// TIA Portal project "Tunel_Paster_16000" (V16)

(* hardware
DEVICE "S7-1200 station_1"  S7-1200 Station
   slot 0: "Rack_0"  S7-1200 Rack  Rack  V1.0
   slot 1: "PLC_1"  CPU 1215C AC/DC/Rly  6ES7 215-1BG40-0XB0  V4.4
*)

// ===== PLC "PLC_1"  CPU 1215C AC/DC/Rly =====

VAR_GLOBAL   // PLC tag table "Default tag table"
   "bStateZones_OK" AT %M10.0 : Bool;   // Все зоны готовы к работе
   "bHasPrior_Stop" AT %M10.1 : Bool;   // Имеется маркер разрешения "СТОП - конвейер
   "bStart_Main_TunelPaster" AT %M1.7 : Bool;   // Старт-Работа тунельного пастеризатора (ОБЩИЙ)
   "bMain_AlarmSystem" AT %M2.3 : Bool;   // АВария в системе (Общая)
   "iNomberZoneAlarm" AT %MW6 : Int;   // Номер зоны с отклонениями
   "Разрешение работы конвейера" AT %M0.0 : Bool;   // Команда разрешения от Глобального блока работы
   "Авария, ошибка в системе" AT %M0.1 : Bool;   // Метка ошибок или аварий
   "Clock_Byte" AT %MB500 : Byte;
   "Clock_10Hz" AT %M500.0 : Bool;
   "Clock_5Hz" AT %M500.1 : Bool;
   "Clock_2.5Hz" AT %M500.2 : Bool;
   "Clock_2Hz" AT %M500.3 : Bool;
   "Clock_1.25Hz" AT %M500.4 : Bool;
   "Clock_1Hz" AT %M500.5 : Bool;
   "Clock_0.625Hz" AT %M500.6 : Bool;
   "Clock_0.5Hz" AT %M500.7 : Bool;
END_VAR

VAR_GLOBAL   // PLC tag table "HMI_"
   "bHMI_button_Start" AT %M2.0 : Bool;   // Кнопка старт
   "bHMI_button_Stop" AT %M2.1 : Bool;   // Кнопка стоп
   "bHMI_button_Pause" AT %M2.2 : Bool;   // Кнопка пауза
   "bHMI_Button_ConveyorStart" AT %M2.4 : Bool;   // Кнопка подтверждения старта конвейера
   "bStartAllowed" AT %M100.0 : Bool;   // Готовность к старту
   "bOpenWindStartConveyor" AT %M100.1 : Bool;   // Вызов окна подтверждения оператором старта конвейера
   "bHMI_ResetAlarm" AT %M0.2 : Bool;   // Сброс аварий
   "iHMI_Num_StatrPaster" AT %MW4 : Int;
   "sHMI_Text_State" AT %MB3 : Char;   // Ткстом статус пастеризатора
   "bTypePID_Zone1" AT %M8.0 : Bool;   // Тип ПИД - 1 - Охлаждение, 0 - Нагрев
   "bTypePID_Zone2" AT %M8.1 : Bool;   // Тип ПИД - 1 - Охлаждение, 0 - Нагрев
   "bTypePID_Zone3" AT %M8.2 : Bool;   // Тип ПИД - 1 - Охлаждение, 0 - Нагрев
   "bTypePID_Zone4" AT %M8.3 : Bool;   // Тип ПИД - 1 - Охлаждение, 0 - Нагрев
   "bTypePID_Zone5" AT %M8.4 : Bool;   // Тип ПИД - 1 - Охлаждение, 0 - Нагрев
END_VAR

VAR_GLOBAL   // PLC tag table "DI"
   "xAlarm_StopButton" AT %I2.0 : Bool;   // Физическая Кнопка стоп
   "xAlarmPump_1" AT %I2.1 : Bool;   // СИгнал аварии от насоса
   "xAlarmPump_2" AT %I2.2 : Bool;   // СИгнал аварии от насоса
   "xAlarmPump_3" AT %I2.3 : Bool;   // СИгнал аварии от насоса
   "xAlarmPump_4" AT %I2.4 : Bool;   // СИгнал аварии от насоса
   "xAlarmPump_5" AT %I2.5 : Bool;   // СИгнал аварии от насоса
   "xAlarmPump_6" AT %I2.6 : Bool;   // СИгнал аварии от насоса
   "xAlarmPump_7" AT %I2.7 : Bool;   // СИгнал аварии от насоса
END_VAR

VAR_GLOBAL   // PLC tag table "Test_PID"
   "set" AT %MD30 : Real;
   "in" AT %MD34 : Real;
   "MAnual" AT %M38.0 : Bool;
   "MValue" AT %MD40 : Real;
   "rOut" AT %MD46 : Real;
   "Mode" AT %MW44 : Int;
   "ResPID" AT %M50.0 : Bool;
END_VAR

VAR_GLOBAL   // PLC tag table "MyTags"
   "InTempZone1" AT %MD12 : Real;   // Зона 1 - температура - обработанная
   "InTempZone2" AT %MD16 : Real;   // Зона 2 - температура - обработанная
   "InTempZone3" AT %MD20 : Real;   // Зона 3 - температура - обработанная
   "InTempZone4" AT %MD24 : Real;   // Зона 4 - температура - обработанная
   "InTempZone5" AT %MD28 : Real;   // Зона 5 - температура - обработанная
END_VAR

TYPE "FV_o/c"
   STRUCT
      bOpenCmd : Bool;   // Команда открыть (автомат)
      bManualMode : Bool;   // Ручной режим (TRUE)
      bManualOpen : Bool;   // Команда открыть в ручном режиме
      bFeedbackOpen : Bool;   // Обратная связь "Открыт"
      tMaxTime : Time;   // Время на открытие
      bResetAlarm : Bool;   // Сброс аварии
      bCheckFeedback : Bool;   // Выбирается есть ли обратная связь у клапана
      bOutOpen : Bool;   // Выход на открытие клапана
      iOutState : Int;   // Выход статуса клапана
      bOutFault : Bool;   // Выход ошибки клапана
   END_STRUCT;
END_TYPE

TYPE "ZoneStatus"
   STRUCT
      bInSetpoint : Bool;   // Зона в уставке по температуре
      bOutOfRange : Bool;   // Зона вышла от уставки на > дельта
      bHasPriority : Bool;   // Зона имеет приоритет на остановку конвейера
   END_STRUCT;
END_TYPE

TYPE "Zone_Pararm"
   STRUCT
      rTemp : Real;   // Температура с датчика
      rSet : Real;   // Уставка
      rDelta : Real;   // Дельта
      bPriority : Bool;   // Приоритет
      bOUT_ZoneStatus : "ZoneStatus";   // Состояние зоны_
   END_STRUCT;
END_TYPE

TYPE "FV_regul"
   STRUCT
      bHMI_ManualMode : Bool;   // Переключение режима авто/ручно (0 - А, 1 - Р)
      rHMI_ManualSet : Real;   // Уставка в ручном режиме (0-100)
      rAuto_Set : Real;   // Уставка в автоматическом режиме
      iOut_AO : Int;   // Сигнал на аналоговый выход
      "rHMI_Out_FV-%" : Real;   // Состояние в % (0-100)
      bOut_DO_ValveOpen : Bool;   // Дискретный сигнал открытия
   END_STRUCT;
END_TYPE

TYPE "Коэф ПИД"
   STRUCT
      Gain : Int;   // Коэф П
      I : DInt;   // Коэф И
      D : DInt;   // Коэф Д
   END_STRUCT;
END_TYPE

TYPE "PE_Param"
   STRUCT
      rСкоростьКонвейера : Real;
      rПЕ_Задан : Real;
      rДлина_Конв : Real;
      rZ_Коэф : Real := 1.393;
      rТref : Real := 60.0;
      rТемп_Мин : Real;
      rТемп_Макс : Real;
      "rСкоростьКонв_м/с" : Real;
      rРучноеЗначТемп : Real;
      diВремяПростоя : DInt := 60000;
      bManualTemp : Bool;
   END_STRUCT;
END_TYPE

// folder: DB-FB

DATA_BLOCK "FB_check_For_Start_DB"   // DB1
{ S7_Optimized_Access := 'FALSE' }
VERSION : 0.1
// stored: InstanceOfName FB_check_For_Start
"FB_check_For_Start"
BEGIN
END_DATA_BLOCK

DATA_BLOCK "FB_Emergency_DB"   // DB3
{ S7_Optimized_Access := 'FALSE' }
VERSION : 0.1
// stored: InstanceOfName -FB_Emergency
"-FB_Emergency"
BEGIN
END_DATA_BLOCK

DATA_BLOCK "FB_CheckZoneStatus_DB"   // DB11
{ S7_Optimized_Access := 'FALSE' }
VERSION : 0.1
// stored: InstanceOfName FB_CheckZoneStatus
"FB_CheckZoneStatus"
BEGIN
END_DATA_BLOCK

DATA_BLOCK "FB_Управление конвейером_DB"   // DB18
{ S7_Optimized_Access := 'FALSE' }
VERSION : 0.1
// stored: InstanceOfName FB_Управление конвейером
"FB_Управление конвейером"
BEGIN
END_DATA_BLOCK

DATA_BLOCK "FB_GlobalStateManager_DB"   // DB31
{ S7_Optimized_Access := 'FALSE' }
VERSION : 0.1
// stored: InstanceOfName FB_GlobalStateManager
"FB_GlobalStateManager"
BEGIN
END_DATA_BLOCK

DATA_BLOCK "FB_PE_Control_DB"   // DB38
{ S7_Optimized_Access := 'TRUE' }
VERSION : 0.1
// stored: InstanceOfName FB_PE_Control
"FB_PE_Control"
BEGIN
END_DATA_BLOCK

// folder: Use VARs to HMI

DATA_BLOCK "DB2_HMI_SET"   // DB2
{ S7_Optimized_Access := 'FALSE' }
VERSION : 0.1
   VAR
      dwSetMinOutDelta : DInt;   // Время ожидания при выходе за пределы уставок
      dwSetMinInDelta : DInt;   // Время ожидания при возврате к уставкам
      dwSetTimeWaitToStart : DInt;   // Время ожидания выхода на режим пастеризатора
      "dwВремя ожидания_стабилизации_темп" : DInt;   // Вреямя ожидания стабилизации температур при выходе за пределы
      rSetTemp_Zone1 : Real;   // Уставка температуры зоны 1
      rSetTemp_Zone2 : Real;   // Уставка температуры зоны 2
      rSetTemp_Zone3 : Real;   // Уставка температуры зоны 3
      rSetTemp_Zone4 : Real;   // Уставка температуры зоны 4
      rSetTemp_Zone5 : Real;   // Уставка температуры зоны 5
      k_PID_Zona1 : "Коэф ПИД";   // ПИД - ЗОна 1
      k_PID_Zona2 : "Коэф ПИД";   // ПИД - зона 2
      k_PID_Zona3 : "Коэф ПИД";   // ПИД - ЗОна 3
      k_PID_Zona4 : "Коэф ПИД";   // ПИД - зона 4
      k_PID_Zona5 : "Коэф ПИД";   // ПИД - ЗОна 5
      HMI_PE : "PE_Param";
   END_VAR
BEGIN
   k_PID_Zona1.Gain := 1;
   k_PID_Zona1.I := 20;
   k_PID_Zona2.Gain := 1;
   k_PID_Zona2.I := 20;
   k_PID_Zona3.Gain := 1;
   k_PID_Zona3.I := 20;
   k_PID_Zona4.Gain := 1;
   k_PID_Zona4.I := 20;
   k_PID_Zona5.Gain := 1;
   k_PID_Zona5.I := 20;
END_DATA_BLOCK

DATA_BLOCK "FVs_o/p"   // DB6
{ S7_Optimized_Access := 'FALSE' }
VERSION : 0.1
   VAR
      FV_1 : "FV_o/c";
      FV_2 : "FV_o/c";
      FV_3 : "FV_o/c";
      FV_4 : "FV_o/c";
      FV_5 : "FV_o/c";
      FV_6 : "FV_o/c";
      FV_7 : "FV_o/c";
   END_VAR
BEGIN
END_DATA_BLOCK

DATA_BLOCK "Zones_Param"   // DB15
{ S7_Optimized_Access := 'FALSE' }
VERSION : 0.1
   VAR
      Zone_1_Преднагрев : "Zone_Pararm";
      Zone_2_Нагрев : "Zone_Pararm";
      Zone_3_Пастеризация : "Zone_Pararm";
      Zone_4_Охлаждение1 : "Zone_Pararm";
      Zone_5_Охлаждение2 : "Zone_Pararm";
   END_VAR
BEGIN
END_DATA_BLOCK

DATA_BLOCK "FVs_Regul"   // DB24
{ S7_Optimized_Access := 'FALSE' }
VERSION : 0.1
   VAR
      FV_Regul_1 : "FV_regul";
      FV_Regul_2 : "FV_regul";
      FV_Regul_3 : "FV_regul";
      FV_Regul_4 : "FV_regul";
      FV_Regul_5 : "FV_regul";
   END_VAR
BEGIN
END_DATA_BLOCK

DATA_BLOCK "Pumps"   // DB30
{ S7_Optimized_Access := 'FALSE' }
VERSION : 0.1
BEGIN
END_DATA_BLOCK

// folder: Зоны/DB_Zone

DATA_BLOCK "FB_Zone_Control_1_Преднагрев_DB"   // DB12
{ S7_Optimized_Access := 'FALSE' }
VERSION : 0.1
// stored: InstanceOfName FB_Zone_Control
"FB_Zone_Control"
BEGIN
END_DATA_BLOCK

DATA_BLOCK "FB_Zone_Control_2_Нагрев_DB"   // DB13
{ S7_Optimized_Access := 'FALSE' }
VERSION : 0.1
// stored: InstanceOfName FB_Zone_Control
"FB_Zone_Control"
BEGIN
END_DATA_BLOCK

DATA_BLOCK "FB_Zone_Control_3_Пастеризация_DB"   // DB14
{ S7_Optimized_Access := 'FALSE' }
VERSION : 0.1
// stored: InstanceOfName FB_Zone_Control
"FB_Zone_Control"
BEGIN
END_DATA_BLOCK

DATA_BLOCK "FB_Zone_Control_4_Охлаждение_DB"   // DB16
{ S7_Optimized_Access := 'FALSE' }
VERSION : 0.1
// stored: InstanceOfName FB_Zone_Control
"FB_Zone_Control"
BEGIN
END_DATA_BLOCK

DATA_BLOCK "FB_Zone_Control_5_Охлаждение2_DB"   // DB17
{ S7_Optimized_Access := 'FALSE' }
VERSION : 0.1
// stored: InstanceOfName FB_Zone_Control
"FB_Zone_Control"
BEGIN
END_DATA_BLOCK

// folder: Клапана/FV_o/C/FV_DB

DATA_BLOCK "FV_1"   // DB4
{ S7_Optimized_Access := 'FALSE' }
VERSION : 0.1
// stored: InstanceOfName Valve(c/o)
"Valve(c/o)"
BEGIN
END_DATA_BLOCK

DATA_BLOCK "FV_5"   // DB5
{ S7_Optimized_Access := 'FALSE' }
VERSION : 0.1
// stored: InstanceOfName Valve(c/o)
"Valve(c/o)"
BEGIN
END_DATA_BLOCK

DATA_BLOCK "FV_6"   // DB7
{ S7_Optimized_Access := 'FALSE' }
VERSION : 0.1
// stored: InstanceOfName Valve(c/o)
"Valve(c/o)"
BEGIN
END_DATA_BLOCK

DATA_BLOCK "FV_7"   // DB8
{ S7_Optimized_Access := 'FALSE' }
VERSION : 0.1
// stored: InstanceOfName Valve(c/o)
"Valve(c/o)"
BEGIN
END_DATA_BLOCK

DATA_BLOCK "FV_2"   // DB9
{ S7_Optimized_Access := 'FALSE' }
VERSION : 0.1
// stored: InstanceOfName Valve(c/o)
"Valve(c/o)"
BEGIN
END_DATA_BLOCK

DATA_BLOCK "FV_3"   // DB10
{ S7_Optimized_Access := 'FALSE' }
VERSION : 0.1
// stored: InstanceOfName Valve(c/o)
"Valve(c/o)"
BEGIN
END_DATA_BLOCK

DATA_BLOCK "FV_4"   // DB19
{ S7_Optimized_Access := 'FALSE' }
VERSION : 0.1
// stored: InstanceOfName Valve(c/o)
"Valve(c/o)"
BEGIN
END_DATA_BLOCK

// folder: Клапана/FV_regul/DB

DATA_BLOCK "FV_Regul_1_DB"   // DB20
{ S7_Optimized_Access := 'FALSE' }
VERSION : 0.1
// stored: InstanceOfName Valve(regul)
"Valve(regul)"
BEGIN
END_DATA_BLOCK

DATA_BLOCK "FV_Regul_2_DB"   // DB21
{ S7_Optimized_Access := 'FALSE' }
VERSION : 0.1
// stored: InstanceOfName Valve(regul)
"Valve(regul)"
BEGIN
END_DATA_BLOCK

DATA_BLOCK "FV_Regul_3_DB"   // DB22
{ S7_Optimized_Access := 'FALSE' }
VERSION : 0.1
// stored: InstanceOfName Valve(regul)
"Valve(regul)"
BEGIN
END_DATA_BLOCK

DATA_BLOCK "FV_Regul_4_DB"   // DB23
{ S7_Optimized_Access := 'FALSE' }
VERSION : 0.1
// stored: InstanceOfName Valve(regul)
"Valve(regul)"
BEGIN
END_DATA_BLOCK

DATA_BLOCK "FV_Regul_5_DB"   // DB37
{ S7_Optimized_Access := 'FALSE' }
VERSION : 0.1
// stored: InstanceOfName Valve(regul)
"Valve(regul)"
BEGIN
END_DATA_BLOCK

// folder: Насосы/DB

DATA_BLOCK "Pump_1_DB"   // DB25
{ S7_Optimized_Access := 'FALSE' }
VERSION : 0.1
// stored: InstanceOfName Pump
"Pump"
BEGIN
END_DATA_BLOCK

DATA_BLOCK "Pump_2_DB"   // DB26
{ S7_Optimized_Access := 'FALSE' }
VERSION : 0.1
// stored: InstanceOfName Pump
"Pump"
BEGIN
END_DATA_BLOCK

DATA_BLOCK "Pump_5_DB"   // DB27
{ S7_Optimized_Access := 'FALSE' }
VERSION : 0.1
// stored: InstanceOfName Pump
"Pump"
BEGIN
END_DATA_BLOCK

DATA_BLOCK "Pump_4_DB"   // DB28
{ S7_Optimized_Access := 'FALSE' }
VERSION : 0.1
// stored: InstanceOfName Pump
"Pump"
BEGIN
END_DATA_BLOCK

DATA_BLOCK "Pump_3_DB"   // DB29
{ S7_Optimized_Access := 'FALSE' }
VERSION : 0.1
// stored: InstanceOfName Pump
"Pump"
BEGIN
END_DATA_BLOCK

// folder: (top level)

FUNCTION_BLOCK "Pump"   // FB1, SCL
{ S7_Optimized_Access := 'FALSE' }
VERSION : 0.1
   VAR_INPUT
      bManualMode : Bool;   // Выбор ручного режима
      bManualStart : Bool;   // Ручной режим - старт
      bManualStop : Bool;   // Ручной режим - стоп
      rManualSpeed : Real;   // Ручной режим - скорость
      bAutoStartPerm : Bool;   // Команда на работоу в авто режиме
      rAutoSpeed : Real;   // Скорость в авто режиме
      bDriveReady : Bool;   // Готовность привода (автоматы)
      bDriveRunning : Bool;   // Привод в работе
      bDriveFault : Bool;   // Привод в ошибке
      rMinSpeed : Real;   // Минимальная скорость
      rMaxSpeed : Real;   // Максимальная скорость
      bResetFault : Bool;   // Сброс аварии
   END_VAR
   VAR_OUTPUT
      bRunCmd : Bool;   // Пуск частотника
      "rSpeedHMI(0-100)" : Real;   // Скорость работы (0-100) для HMI
      iSpeedOut : Int;   // Скорость насоса для аналогового выхода
      bPumpRunning : Bool;   // Работа
      bPumpFault : Bool;   // Авария
      iStatus : Int;   // Статус (0 - стоп 1 - работа 2 - авария)
   END_VAR
   VAR
      bFaultLatch : Bool;
      bRunRequest : Bool;
      rSpeedPump : Real;   // Скорость насоса
   END_VAR
BEGIN
   // 1. Обработка аварий
   #bFaultLatch := (#bDriveFault OR #bFaultLatch) AND NOT #bResetFault;
   #bPumpFault := #bFaultLatch;

   // 2. Формирование команды "Пуск"
   IF #bManualMode THEN
       // Ручной режим
       IF #bManualStart AND NOT #bManualStop THEN
           #bRunRequest := TRUE;
       ELSIF #bManualStop OR NOT #bDriveReady THEN
           #bRunRequest := FALSE;
       END_IF;
   ELSE
       // Автоматический режим
       #bRunRequest := #bAutoStartPerm AND NOT #bDriveFault;
   END_IF;

   // 3. Задание скорости
   IF #bManualMode THEN
       #"rSpeedHMI(0-100)" := LIMIT(MN := #rMinSpeed, IN := #rManualSpeed, MX := #rMaxSpeed);
   ELSE
       #"rSpeedHMI(0-100)" := LIMIT(MN := #rMinSpeed, IN := #rAutoSpeed, MX := #rMaxSpeed);
   END_IF;

   // Преобразование значения от 0-100 до 0-27648 для аналогового выхода
   #iSpeedOut := REAL_TO_INT((#"rSpeedHMI(0-100)"/ 100.0) * 27648.0);

   // 4. Выходные команды и статусы
   #bRunCmd := #bRunRequest AND NOT #bFaultLatch AND #bDriveReady;
   #bPumpRunning := #bDriveRunning AND #bRunCmd;

   // 5. Числовой статус (для HMI/SCADA)
   IF #bFaultLatch THEN
       #iStatus := 2; // Авария
   ELSIF #bPumpRunning THEN
       #iStatus := 1; // Работа
   ELSE
       #iStatus := 0; // Стоп
   END_IF;
END_FUNCTION_BLOCK

FUNCTION_BLOCK "FB_GlobalStateManager"   // FB2, SCL
{ S7_Optimized_Access := 'FALSE' }
VERSION : 0.1
   VAR_INPUT
      bStartCmd : Bool;   // Команда на старт от HMI
      bConfirmStart : Bool;   // Подтверждение оператора
      bResetFault : Bool;   // Сброс ошибки
      bAllSetpointsReached : Bool;   // // Все температуры достигли уставок
      bNoFaults : Bool;   // Нет аварий
      tStartTimeout : Time := T#30m;   // Время за которое пастер выходит на режим
      tReadyDelay : Time := t#10s;   // Время ожидания при выходе на режим до готовности
   END_VAR
   VAR_OUTPUT
      eState : Int;   // Текущее состояние
      bConveyorEnable : Bool;   // Разрешение на работу конвейера
      bSystemReady : Bool;   // Готовность системы
      bSystemFault : Bool;   // Состояние Fault
      sStatusText : WString;   // Текст для HMI
   END_VAR
   VAR
      tonStartTimeout : TON_TIME;   // Таймер выхода на режим
      tonReadyDelay : TON_TIME;   // Таймер готовности
   END_VAR
   VAR CONSTANT
      cSTATE_IDLE : Int;
      cSTATE_CHECK : Int := 10;
      cSTATE_STARTING : Int := 20;
      cSTATE_READY_DELAY : Int := 30;
      cSTATE_READY : Int := 40;
      cSTATE_FAULT : Int := 99;
      sText1 : String := 'Waiting';
   END_VAR
BEGIN
   // Таймеры
   #tonStartTimeout(IN := (#eState = #cSTATE_STARTING) AND NOT #bAllSetpointsReached, PT := #tStartTimeout);

   #tonReadyDelay(IN := (#eState = #cSTATE_READY_DELAY), PT := #tReadyDelay);

   // Основной CASE
   CASE #eState OF

       #cSTATE_IDLE:
        //   #sStatusText := 'Ожидание команды старта';
           IF #bStartCmd THEN
               #eState := #cSTATE_CHECK;
           END_IF;

       #cSTATE_CHECK:
       //    #sStatusText := 'Проверка условий старта';
           IF NOT #bNoFaults THEN
               #eState := #cSTATE_FAULT;
           ELSE
               #eState := #cSTATE_STARTING;
           END_IF;

       #cSTATE_STARTING:
      //     #sStatusText := 'Выход на уставки';
           IF #bAllSetpointsReached THEN
               #eState := #cSTATE_READY_DELAY;
           ELSIF #tonStartTimeout.Q THEN
               #eState := #cSTATE_FAULT;
           END_IF;

       #cSTATE_READY_DELAY:
      //     #sStatusText := 'dfsf';
           IF #tonReadyDelay.Q THEN
               #eState := #cSTATE_READY_DELAY;
           END_IF;

       #cSTATE_READY_DELAY:
      //     #sStatusText := 'Готово, ожидание подтверждения';
           #bSystemReady := TRUE;
           IF #bConfirmStart THEN
               #bConveyorEnable := TRUE;
           END_IF;

       #cSTATE_FAULT:
     //      #sStatusText := 'Авария! Требуется сброс';
           #bSystemFault := TRUE;
           IF #bResetFault AND #bNoFaults THEN
               #eState := #cSTATE_IDLE;
           END_IF;

       ELSE
           #eState := #cSTATE_IDLE;

   END_CASE;
END_FUNCTION_BLOCK

FUNCTION_BLOCK "Valve(c/o)"   // FB3, SCL
{ S7_Optimized_Access := 'FALSE' }
VERSION : 0.1
   VAR_INPUT
      bAuto_OpenCmd : Bool;   // Команда открыть (автомат)
      bManualMode : Bool;   // Ручной режим (TRUE)
      bManualOpen : Bool;   // Команда открыть в ручном режиме
      bFeedbackOpen : Bool;   // Обратная связь "Открыт"
      tMaxTime : Time;   // Время на открытие
      bResetAlarm : Bool;   // Сброс аварии
      bHaveFeedback : Bool;   // Есть ли обратная связь (0 - нет, 1 есть)
   END_VAR
   VAR_OUTPUT
      bValveOpen : Bool;   // Управляющий выход
      iValveState : Int;   // 0 = Закрыт, 1 = Открыт, 2 = Авария
      bValveFault : Bool;   // Авария
   END_VAR
   VAR
      tiOpenTimer : TON_TIME;   // Таймер на открытие
      bWaitingOpen : Bool;   // Флаг ожидания открытия
      bEnableTimer : Bool;   // Флаг активации таймера
   END_VAR
BEGIN

   // Обновление таймера — всегда в одном месте, вне условий
   #tiOpenTimer(
                IN := #bEnableTimer,
                PT := #tMaxTime
   );

   // Сброс
   IF #bResetAlarm THEN
       #bValveFault := FALSE;
       #bWaitingOpen := FALSE;
       #bEnableTimer := FALSE;
   END_IF;

   // === Режим: РУЧНОЙ ===
   IF #bManualMode THEN
       #bValveOpen := #bManualOpen;
       #bValveFault := FALSE;          // Аварии в ручном режиме не учитываются
       #bEnableTimer := FALSE;
       #bWaitingOpen := FALSE;

       // === Режим: АВТО ===
   ELSE

           // Управление выходом с учетом аварии, с контролем обратной связи
        IF #bAuto_OpenCmd AND NOT #bValveFault THEN
                   #bValveOpen := TRUE;
        ELSE
                   #bValveOpen := FALSE;
               END_IF;

               //  Проверяем, есть ли контроль обратной связи
        IF #bHaveFeedback THEN
            // Контроль открытия
            IF #bAuto_OpenCmd AND NOT #bFeedbackOpen AND NOT #bValveFault THEN
                #bEnableTimer := TRUE;
                #bWaitingOpen := TRUE;
            ELSE
                #bEnableTimer := FALSE;
                ;
                IF #bFeedbackOpen THEN
                    #bWaitingOpen := FALSE;
                END_IF;
            END_IF;
        END_IF;


           // Авария
           IF #tiOpenTimer.Q AND #bWaitingOpen THEN
               #bValveFault := TRUE;
               #bWaitingOpen := FALSE;
           END_IF;

   END_IF;


   // Состояние клапана
   IF #bValveFault THEN
       #iValveState := 2;       // Авария
   ELSIF #bHaveFeedback AND #bFeedbackOpen  THEN
       #iValveState := 1;       // Открыт
   ELSIF NOT #bHaveFeedback AND (NOT #bManualMode AND #bAuto_OpenCmd) OR (#bManualOpen AND #bManualMode) THEN
       #iValveState := 1;       // Открыт 
   ELSE
       #iValveState := 0;       // Закрыт
   END_IF;
END_FUNCTION_BLOCK

FUNCTION_BLOCK "Valve(regul)"   // FB4, SCL
{ S7_Optimized_Access := 'FALSE' }
VERSION : 0.1
   VAR_INPUT
      bManualMode : Bool;   // TRUE = ручной режим, FALSE = автоматический режим
      rAutoSetpoint : Real;   // Уставка открытия клапана в % (0.0–100.0) в автомате
      rManualSetpoint : Real;   // Уставка открытия клапана в % (0.0–100.0) в ручном режиме
   END_VAR
   VAR_OUTPUT
      iAnalogOutput : Int;   // Значение для аналогового выхода (0–27648)
      rValvePosPercent : Real;   // Текущее % открытия клапана для HMI
      bValveOpen : Bool;   // Дискретный сигнал "клапан открыт" (TRUE, если >0%)
   END_VAR
   VAR
      rSetpointPercent : Real;   // Расчётная уставка % открытия в текущем режиме
   END_VAR
BEGIN
       // Выбор уставки в зависимости от режима
       IF #bManualMode THEN
           #rSetpointPercent := #rManualSetpoint;
       ELSE
           #rSetpointPercent := #rAutoSetpoint;
       END_IF;

       // Ограничение % от 0.0 до 100.0
       IF #rSetpointPercent < 0.0 THEN
           #rSetpointPercent := 0.0;
       ELSIF #rSetpointPercent > 100.0 THEN
           #rSetpointPercent := 100.0;
       END_IF;

       // Перевод % в значение для аналогового выхода
       #iAnalogOutput := REAL_TO_INT((#rSetpointPercent / 100.0) * 27648.0);

           // Вывод значения для HMI
       #rValvePosPercent := #rSetpointPercent;

       // Дискретный сигнал "клапан открыт", если % > 0
       #bValveOpen := #rSetpointPercent > 0.0;
END_FUNCTION_BLOCK

FUNCTION_BLOCK "FB_Управление конвейером"   // FB5, SCL
{ S7_Optimized_Access := 'FALSE' }
VERSION : 0.1
   VAR_INPUT
      bEnable : Bool;   // Общий флаг работы системы
      bStartCmd : Bool;   // Команда на запуск от HMI, по кнопке из окна подтверждения
      bAllZonesInSetpoint : Bool;   // Все зоны достигли уставок
      bGlobalFault : Bool;   // Авария по системе
      bZoneHasPriority : Bool;   // У зоны с отклонением есть приоритет
      dwDeltaTempDelayMin : DWord;   // Задержка (мин), прежде чем остановить конвейер при отклонении
      dwResumeDelayMin : DInt;   // Время возврата после нормализации
   END_VAR
   VAR_OUTPUT
      bConveyorRun : Bool;   // Команда на пуск частотников
      bReadyToStart : Bool;   // Готовность к работе конвейера
      bWaitingConfirm : Bool;   // Ждём подтверждения от оператора, вывод окна на HMI
      bPaused : Bool;   // Конвейер остановлен по отклонению
   END_VAR
   VAR
      bStarted : Bool;   // Внутреннее состояние — процесс стартовал
      tiPauseTimer : TON_TIME;   // Таймер задержки перед остановкой
      tiResumeTimer : TON_TIME;   // Таймер ожидания перед возобновлением
      aZoneS_Status : Array[1..5] of "ZoneStatus";   // Массив для сбора состояния зон
      i : Int;
   END_VAR
   // tiPauseTimer.PT := T#1s;
   // tiResumeTimer.PT := T#1s;
BEGIN

   // Проверка на наличие флага обей работы системы
   IF NOT #bEnable THEN
       #bReadyToStart := FALSE;
       #bWaitingConfirm := FALSE;
       #bConveyorRun := FALSE;
       #bPaused := FALSE;
       #tiPauseTimer.IN := FALSE;
       #tiResumeTimer.IN := FALSE;
       RETURN;
   END_IF;



   // Условия готовности к запуску
   IF NOT #bStarted AND NOT #bGlobalFault AND #bAllZonesInSetpoint THEN
       #bReadyToStart := TRUE;

           // Команда на старт — вручную подтверждена
           IF NOT #bStartCmd THEN
               #bWaitingConfirm := TRUE;
           END_IF;

   ELSE
       #bReadyToStart := FALSE;
       #bWaitingConfirm := FALSE;
   END_IF;



   IF #bStartCmd AND #bReadyToStart THEN
       #bStarted := TRUE;
       #bWaitingConfirm := FALSE;
   END_IF;

   // После старта разрешаем работу, если нет аварий и температур в норме
   IF #bStarted AND NOT #bGlobalFault THEN

       IF NOT #bAllZonesInSetpoint THEN
           IF #bZoneHasPriority THEN
               // Включаем таймер паузы, задержка перед остановкой
               #tiPauseTimer(IN := TRUE,
                             PT := (#dwDeltaTempDelayMin * 60000)) //В минутах
               ;
           ELSE
               #tiPauseTimer(IN := FALSE,PT := t#0s);
           END_IF;

           // Переход в паузу
           IF #tiPauseTimer.Q THEN
               #bPaused := TRUE;
               #bConveyorRun := FALSE;
               #tiResumeTimer(IN := FALSE, PT := t#0s); // Сброс таймера возобновления

           END_IF;

       ELSE
           // Температуры вернулись в норму — запускаем таймер на возврат
           IF #bPaused THEN
               #tiResumeTimer(IN := TRUE,
                              PT := (#dwResumeDelayMin * 60000)) // в минутах
               ;
               // Возвращаемся к работе
               IF #tiResumeTimer.Q THEN
                   #bPaused := FALSE;
                   #bConveyorRun := TRUE;
                   #tiResumeTimer(IN := FALSE, PT := t#0s); // сброс таймера
               END_IF;
           ELSE
               #bConveyorRun := TRUE;
               #tiPauseTimer(IN := FALSE, PT := t#0s); // сброс
               #tiResumeTimer(IN := FALSE,PT := t#0s);
           END_IF;
       END_IF;
   ELSE
       // Если глобальная авария — всё стоп
       #bConveyorRun := FALSE;
       #bPaused := FALSE;
       #bStarted := FALSE;
       #tiPauseTimer(IN := FALSE, PT := t#0s);
       #tiResumeTimer(IN := FALSE,PT := t#0s);
       #bWaitingConfirm := FALSE;
   END_IF;
END_FUNCTION_BLOCK

FUNCTION_BLOCK "FB_Motor_Conveyor"   // FB6, SCL
{ S7_Optimized_Access := 'FALSE' }
VERSION : 0.1
   VAR_INPUT
      bManualMode : Bool;   // Выбор ручного режима
      bManualStart : Bool;   // Ручной режим - старт
      bManualStop : Bool;   // Ручной режим - стоп
      rManualSpeed : Real;   // Ручной режим - скорость
      bAutoStartPerm : Bool;   // Команда на работоу в авто режиме
      rAutoSpeed : Real;   // Скорость в авто режиме
      bDriveReady : Bool;   // Готовность привода (автоматы)
      bDriveRunning : Bool;   // Привод в работе
      bDriveFault : Bool;   // Привод в ошибке
      rMinSpeed : Real;   // Минимальная скорость
      rMaxSpeed : Real;   // Максимальная скорость
      bResetFault : Bool;   // Сброс аварии
   END_VAR
   VAR_OUTPUT
      bRunCmd : Bool;   // Пуск частотника
      "rSpeedHMI(0-100)" : Real;   // Скорость работы (0-100) для HMI
      iSpeedOut : Int;   // Скорость насоса для аналогового выхода
      bPumpRunning : Bool;   // Работа
      bPumpFault : Bool;   // Авария
      iStatus : Int;   // Статус (0 - стоп 1 - работа 2 - авария)
   END_VAR
   VAR
      bFaultLatch : Bool;
      bRunRequest : Bool;
      rSpeedPump : Real;   // Скорость насоса
   END_VAR
BEGIN
   // 1. Обработка аварий
   #bFaultLatch := (#bDriveFault OR #bFaultLatch) AND NOT #bResetFault;
   #bPumpFault := #bFaultLatch;

   // 2. Формирование команды "Пуск"
   IF #bManualMode THEN
       // Ручной режим
       IF #bManualStart AND NOT #bManualStop THEN
           #bRunRequest := TRUE;
       ELSIF #bManualStop OR NOT #bDriveReady THEN
           #bRunRequest := FALSE;
       END_IF;
   ELSE
       // Автоматический режим
       #bRunRequest := #bAutoStartPerm AND NOT #bDriveFault;
   END_IF;

   // 3. Задание скорости
   IF #bManualMode THEN
       #"rSpeedHMI(0-100)" := LIMIT(MN := #rMinSpeed, IN := #rManualSpeed, MX := #rMaxSpeed);
   ELSE
       #"rSpeedHMI(0-100)" := LIMIT(MN := #rMinSpeed, IN := #rAutoSpeed, MX := #rMaxSpeed);
   END_IF;

   // Преобразование значения от 0-100 до 0-27648 для аналогового выхода
   #iSpeedOut := REAL_TO_INT((#"rSpeedHMI(0-100)"/ 100.0) * 27648.0);

   // 4. Выходные команды и статусы
   #bRunCmd := #bRunRequest AND NOT #bFaultLatch AND #bDriveReady;
   #bPumpRunning := #bDriveRunning AND #bRunCmd;

   // 5. Числовой статус (для HMI/SCADA)
   IF #bFaultLatch THEN
       #iStatus := 2; // Авария
   ELSIF #bPumpRunning THEN
       #iStatus := 1; // Работа
   ELSE
       #iStatus := 0; // Стоп
   END_IF;
END_FUNCTION_BLOCK

FUNCTION_BLOCK "-FB_Emergency"   // FB7, SCL
{ S7_Optimized_Access := 'FALSE' }
VERSION : 0.1
   VAR_INPUT
      EmergencyStopButton : Bool;   // Аварийный стоп-кнопка
      PumpFault : Bool;   // Авария насосов
      ValveFault : Bool;   // Авария клапанов
      LongWarmUpFault : Bool;   // Долгий выход на режим
      ProductStuck : Bool;   // Застревание продукции
      ResetEmergency : Bool;   // Сброс аварии (кнопка на панели/системе)
   END_VAR
   VAR_OUTPUT
      EmergencyActive : Bool;   // Флаг активной аварии
      EmergencyCode : Int;   // Код аварии для отображения на HMI
   END_VAR
   VAR
      LatchedEmergency : Bool;   // Зафиксированная аварийная ситуация
      InternalCode : Bool;   // Внутренний код аварии
   END_VAR
BEGIN
   #EmergencyCode := 0;
   IF #EmergencyStopButton THEN
       #EmergencyCode := #EmergencyCode OR 2#00000001; // Бит 0
   END_IF;
   IF #PumpFault THEN
       #EmergencyCode := #EmergencyCode OR 2#00000010; // Бит 1
   END_IF;
   IF #ValveFault THEN
       #EmergencyCode := #EmergencyCode OR 2#00000100; // Бит 2
   END_IF;
   IF #LongWarmUpFault THEN
       #EmergencyCode := #EmergencyCode OR 2#00001000; // Бит 3
   END_IF;
   IF #ProductStuck THEN
       #EmergencyCode := #EmergencyCode OR 2#00010000; // Бит 4
   END_IF;

   // Считаем, что авария активна, если хоть один бит установлен
   #EmergencyActive := #EmergencyCode <> 0;

   // Сброс аварии
   IF #ResetEmergency THEN
       #EmergencyCode := 0;
       #EmergencyActive := FALSE;
   END_IF;
END_FUNCTION_BLOCK

FUNCTION_BLOCK "FB_Zone_Control"   // FB8, SCL
{ S7_Optimized_Access := 'FALSE' }
VERSION : 0.1
   VAR_INPUT
      rTempActual : Real;   // Температура с датчика
      rTempSetpoint : Real;   // Уставка температуры
      rDelta : Real;   // Допустимое отклонение от уставки
      bPriority : Bool;   // Приоритет управления конвейером (1 - стоп конвейер)
   END_VAR
   VAR_OUTPUT
      ZoneStatusOut : "ZoneStatus";
      bInSetpoint : Bool;
      bOutOfRange : Bool;
      bHasPriority : Bool;
   END_VAR
BEGIN
   // ---------- Реализация логики зоны ----------
   // 
                       // --------Проверка зоны что в уставке---------
           #ZoneStatusOut.bInSetpoint := ABS(#rTempActual - #rTempSetpoint) <= #rDelta;

           // --------Проверка зоны что вышла за уставку---------
           #ZoneStatusOut.bOutOfRange := ABS(#rTempActual - #rTempSetpoint) > #rDelta;

           // -------Проверяем преоритет зоны-------
           #ZoneStatusOut.bHasPriority := #bPriority;


           //---Статусы отдельными выходами, для наглядности-----
           //
           #bInSetpoint := #ZoneStatusOut.bInSetpoint;
           #bOutOfRange := #ZoneStatusOut.bOutOfRange;
           #bHasPriority := #bPriority;
END_FUNCTION_BLOCK

FUNCTION_BLOCK "FB_check_For_Start"   // FB9, SCL
{ S7_Optimized_Access := 'FALSE' }
VERSION : 0.1
   VAR_INPUT
      xHMI_Start : Bool;   // кнопка старта с HMI
      xEmergency_Stop : Bool;   // аварийный стоп
      xSystem_Ready : Bool;   // Готовность всех систем
      xStopHMI : Bool;   // Кнопка СТОП на HMI
   END_VAR
   VAR_OUTPUT
      xStart_Allowed : Bool;   // Разрешение на РАБОТУ
      xStart : Bool;   // Работа пастеризатора
   END_VAR
   VAR
      "m" : Bool;   // memory
   END_VAR
BEGIN

   //Проверка на разрешение работы.
   //
   IF NOT #xEmergency_Stop AND #xSystem_Ready THEN
       #xStart_Allowed := TRUE;
   ELSE
       #xStart_Allowed := FALSE;
   END_IF;

   #xStart := (#xStart OR #xHMI_Start) AND NOT (#xEmergency_Stop OR #xStopHMI);
END_FUNCTION_BLOCK

FUNCTION_BLOCK "FB_CheckZoneStatus"   // FB10, SCL
{ S7_Optimized_Access := 'FALSE' }
VERSION : 0.1
   VAR_OUTPUT
      bAllZones_Redy : Bool;   // Выход состояния всех зон ОК
      bPriority_Stop : Bool;   // Выход 1 - если есть метка остановки конвейера
      iZonesNumberFail : Int;   // ВЫход с Номером зоны
   END_VAR
   VAR
      aZoneS_Status : Array[1..5] of "ZoneStatus";   // Массив с данными по всем зонам
      i : Int;
      AllZone_Ok : Bool;   // Состояние всех зон ОК
      HaveStopPriority : Bool;   // В зоне есть метка для остановки конвейера
      iNumber : Int;   // Номер зоны, где отклонение температуры
   END_VAR
BEGIN


           // ----Сбор данных по всем зонам в массив для обработки-----
   #aZoneS_Status[1] := "Zones_Param".Zone_1_Преднагрев.bOUT_ZoneStatus;
   #aZoneS_Status[2] := "Zones_Param".Zone_2_Нагрев.bOUT_ZoneStatus;
   #aZoneS_Status[3] := "Zones_Param".Zone_3_Пастеризация.bOUT_ZoneStatus;
   #aZoneS_Status[4] := "Zones_Param".Zone_4_Охлаждение1.bOUT_ZoneStatus;
   #aZoneS_Status[5] := "Zones_Param".Zone_5_Охлаждение2.bOUT_ZoneStatus;

           //Сброс маркеров по умолчанию----
   #AllZone_Ok := TRUE;    
   #HaveStopPriority := FALSE;
   #iNumber := 0;
              // ----Цикл для перебора всех зон значение выставить по количеству зон----
   FOR #i := 1 TO 5 DO
       IF NOT #aZoneS_Status[#i].bInSetpoint THEN
           #AllZone_Ok := FALSE;
           #iNumber := #i;
           IF #aZoneS_Status[#i].bHasPriority THEN
               #HaveStopPriority := TRUE;
           END_IF;
       END_IF;
   END_FOR;

   /// Присвоение переменных к выходам
   #bAllZones_Redy := #AllZone_Ok;
   #bPriority_Stop := #HaveStopPriority;
   #iZonesNumberFail := #iNumber;
END_FUNCTION_BLOCK

FUNCTION_BLOCK "FB_PE_Control"   // FB11, SCL
{ S7_Optimized_Access := 'TRUE' }
VERSION : 0.1
   VAR_INPUT
      bRunRequest : Bool;   // Запрос на работу
      rSpeedPercent : Real;   // Заданная скорость от оператора (0…100%)
      rPESetpoint : Real;   // Заданное количество ПЕ
      rConveyorLength : Real;   // Длина зоны выдержки, м
      rZParam : Real;   // Коэффициент z (1.393 обычно)
      rTref : Real;   // Температура при которой 1 ПЕ за 1 мин (обычно 60°C)
      rTmin : Real;   // Мин допустимая температура
      rTmax : Real;   // Макс допустимая температура
      rVmax : Real;   // акс скорость м/с (например 0.2 м/с)
      bManualMode : Bool;   // Режим "ручной расчёт температуры"
      rManualTemp : Real;   // Температура в ручном режиме
      bAlarm : Bool;   // Общая авария
      tStopTolerance : Time;   // Допустимое время простоя
   END_VAR
   VAR_OUTPUT
      rTempSetpoint : Real;   // Уставка температуры
      rHoldTime : Real;   // Время выдержки в секундах
      rConveyorSpeed : Real;   // Скорость конвейера (м/с)
      bTempValid : Bool;   // Температура в пределах допустимого
      bAlarmHigh : Bool;   // Температура превышает максимум
      bAlarmLow : Bool;   // Температура ниже минимума
      bStoppedTooLong : Bool;   // Превышено время простоя
      bAlarmTempOverride : Bool;   // Принудительная уставка из-за аварии
   END_VAR
   VAR RETAIN
      rSpeedRatio : Real;   // Отношение скорости
      rPENeededPerMin : Real;   // Требуемое ПЕ в минуту
      rLogArg : Real;   // Аргумент логарифма
   END_VAR
   VAR
      TON_StopDelay : TON_TIME;   // Таймер задержки останова
   END_VAR
BEGIN
   // Блок управления уставкой температуры по ПЕ и скорости
   // Сначала сброс в случае остановки
   IF NOT #bRunRequest THEN
       #rTempSetpoint := 0.0;
       #rHoldTime := 0.0;
       #rConveyorSpeed := 0.0;
       #bTempValid := TRUE;
       #bAlarmHigh:= FALSE;
       #bAlarmLow := FALSE;
       #bAlarmTempOverride := FALSE;
       #bStoppedTooLong := FALSE;
       #TON_StopDelay(IN := FALSE, PT := t#0s);
       RETURN;
   END_IF;


   // Преобразуем % скорости в отношение
   #rSpeedRatio := #rSpeedPercent / 100.0;

   // Расчёт фактической скорости (м/с)
   #rConveyorSpeed := #rVmax * #rSpeedRatio;

   // Время нахождения бутылки в зоне (сек)
   IF #rConveyorSpeed > 0.0 THEN
       #rHoldTime := #rConveyorLength / #rConveyorSpeed; // В секундах
   ELSE
       #rHoldTime := 0.0;
   END_IF;


   IF #bManualMode THEN
       // Ручной режим — берём температуру с панели
       #rTempSetpoint := #rManualTemp;
   ELSE
       // Расчёт температуры по ПЕ
       IF #rHoldTime > 0.0 AND #rPESetpoint > 0.0 THEN
           #rPENeededPerMin := #rPESetpoint * 60.0 / #rHoldTime;
           #rLogArg := LN(#rPENeededPerMin) / LN(10.0);
           #rTempSetpoint := #rTref + #rLogArg / #rZParam;
       ELSE
           #rTempSetpoint := #rTref; // по умолчанию
       END_IF;
   END_IF;

   // Проверка пределов
   #bTempValid := TRUE;
   #bAlarmHigh := FALSE;
   #bAlarmLow := FALSE;


   IF #rTempSetpoint > #rTmax THEN
       #rTempSetpoint := #rTmax;
       #bTempValid := FALSE;
       #bAlarmHigh := TRUE;
   ELSIF #rTempSetpoint < #rTmin THEN
       #rTempSetpoint := #rTmin;
       #bTempValid := FALSE;
       #bAlarmLow := TRUE;
   END_IF;
END_FUNCTION_BLOCK

FUNCTION "Клапана_О/З" : Void   // FC1, LAD
{ S7_Optimized_Access := 'TRUE' }
VERSION : 0.1
BEGIN

REGION Network 1: FV-1
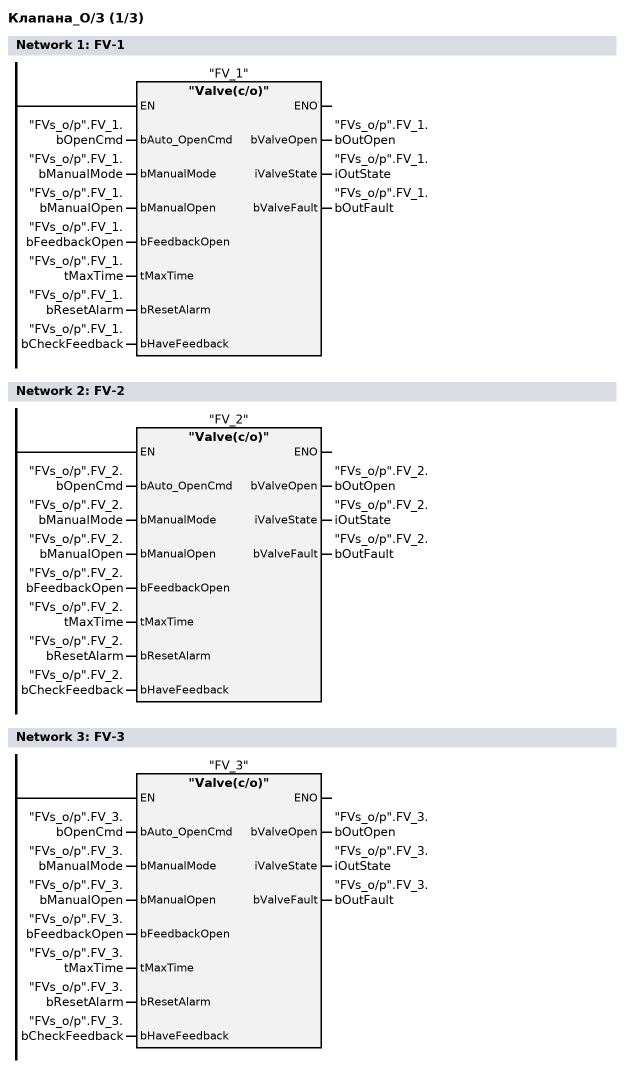
   RUNG wire#powerrail
      "FV_1"(bAuto_OpenCmd := "FVs_o/p".FV_1.bOpenCmd, bManualMode := "FVs_o/p".FV_1.bManualMode, bManualOpen := "FVs_o/p".FV_1.bManualOpen, bFeedbackOpen := "FVs_o/p".FV_1.bFeedbackOpen, tMaxTime := "FVs_o/p".FV_1.tMaxTime, bResetAlarm := "FVs_o/p".FV_1.bResetAlarm, bHaveFeedback := "FVs_o/p".FV_1.bCheckFeedback, bValveOpen => "FVs_o/p".FV_1.bOutOpen, iValveState => "FVs_o/p".FV_1.iOutState, bValveFault => "FVs_o/p".FV_1.bOutFault)
   END_RUNG
   // the same network as SCL:
   "FV_1"(bAuto_OpenCmd := "FVs_o/p".FV_1.bOpenCmd,   // "Valve(c/o)"
          bManualMode := "FVs_o/p".FV_1.bManualMode,
          bManualOpen := "FVs_o/p".FV_1.bManualOpen,
          bFeedbackOpen := "FVs_o/p".FV_1.bFeedbackOpen,
          tMaxTime := "FVs_o/p".FV_1.tMaxTime,
          bResetAlarm := "FVs_o/p".FV_1.bResetAlarm,
          bHaveFeedback := "FVs_o/p".FV_1.bCheckFeedback,
          bValveOpen => "FVs_o/p".FV_1.bOutOpen,
          iValveState => "FVs_o/p".FV_1.iOutState,
          bValveFault => "FVs_o/p".FV_1.bOutFault);
END_REGION

REGION Network 2: FV-2
   RUNG wire#powerrail
      "FV_2"(bAuto_OpenCmd := "FVs_o/p".FV_2.bOpenCmd, bManualMode := "FVs_o/p".FV_2.bManualMode, bManualOpen := "FVs_o/p".FV_2.bManualOpen, bFeedbackOpen := "FVs_o/p".FV_2.bFeedbackOpen, tMaxTime := "FVs_o/p".FV_2.tMaxTime, bResetAlarm := "FVs_o/p".FV_2.bResetAlarm, bHaveFeedback := "FVs_o/p".FV_2.bCheckFeedback, bValveOpen => "FVs_o/p".FV_2.bOutOpen, iValveState => "FVs_o/p".FV_2.iOutState, bValveFault => "FVs_o/p".FV_2.bOutFault)
   END_RUNG
   // the same network as SCL:
   "FV_2"(bAuto_OpenCmd := "FVs_o/p".FV_2.bOpenCmd,   // "Valve(c/o)"
          bManualMode := "FVs_o/p".FV_2.bManualMode,
          bManualOpen := "FVs_o/p".FV_2.bManualOpen,
          bFeedbackOpen := "FVs_o/p".FV_2.bFeedbackOpen,
          tMaxTime := "FVs_o/p".FV_2.tMaxTime,
          bResetAlarm := "FVs_o/p".FV_2.bResetAlarm,
          bHaveFeedback := "FVs_o/p".FV_2.bCheckFeedback,
          bValveOpen => "FVs_o/p".FV_2.bOutOpen,
          iValveState => "FVs_o/p".FV_2.iOutState,
          bValveFault => "FVs_o/p".FV_2.bOutFault);
END_REGION

REGION Network 3: FV-3
   RUNG wire#powerrail
      "FV_3"(bAuto_OpenCmd := "FVs_o/p".FV_3.bOpenCmd, bManualMode := "FVs_o/p".FV_3.bManualMode, bManualOpen := "FVs_o/p".FV_3.bManualOpen, bFeedbackOpen := "FVs_o/p".FV_3.bFeedbackOpen, tMaxTime := "FVs_o/p".FV_3.tMaxTime, bResetAlarm := "FVs_o/p".FV_3.bResetAlarm, bHaveFeedback := "FVs_o/p".FV_3.bCheckFeedback, bValveOpen => "FVs_o/p".FV_3.bOutOpen, iValveState => "FVs_o/p".FV_3.iOutState, bValveFault => "FVs_o/p".FV_3.bOutFault)
   END_RUNG
   // the same network as SCL:
   "FV_3"(bAuto_OpenCmd := "FVs_o/p".FV_3.bOpenCmd,   // "Valve(c/o)"
          bManualMode := "FVs_o/p".FV_3.bManualMode,
          bManualOpen := "FVs_o/p".FV_3.bManualOpen,
          bFeedbackOpen := "FVs_o/p".FV_3.bFeedbackOpen,
          tMaxTime := "FVs_o/p".FV_3.tMaxTime,
          bResetAlarm := "FVs_o/p".FV_3.bResetAlarm,
          bHaveFeedback := "FVs_o/p".FV_3.bCheckFeedback,
          bValveOpen => "FVs_o/p".FV_3.bOutOpen,
          iValveState => "FVs_o/p".FV_3.iOutState,
          bValveFault => "FVs_o/p".FV_3.bOutFault);
END_REGION

REGION Network 4: FV-4
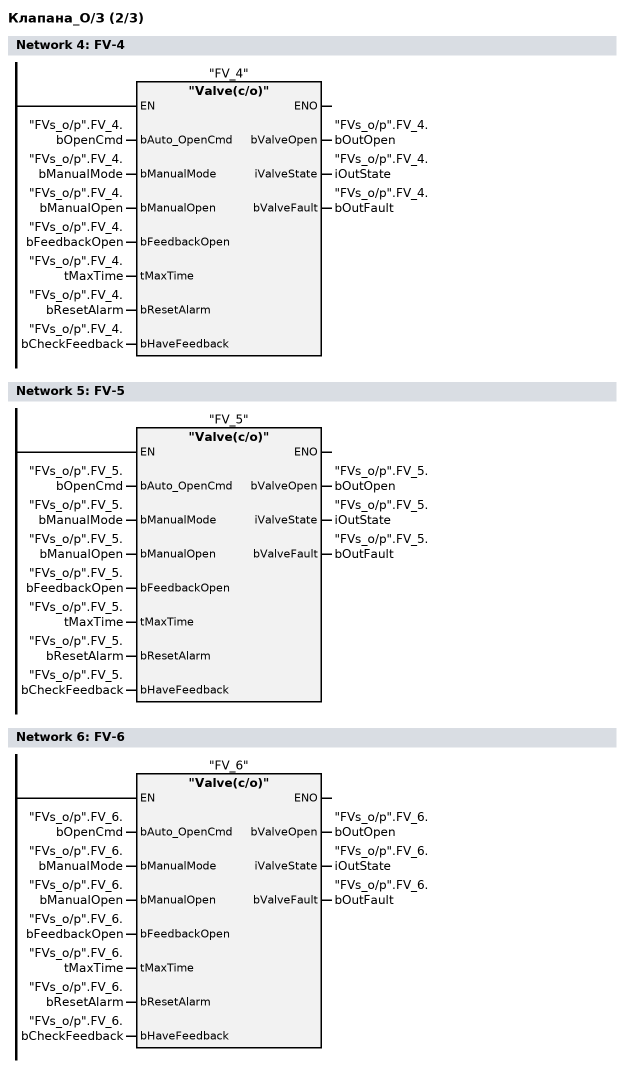
   RUNG wire#powerrail
      "FV_4"(bAuto_OpenCmd := "FVs_o/p".FV_4.bOpenCmd, bManualMode := "FVs_o/p".FV_4.bManualMode, bManualOpen := "FVs_o/p".FV_4.bManualOpen, bFeedbackOpen := "FVs_o/p".FV_4.bFeedbackOpen, tMaxTime := "FVs_o/p".FV_4.tMaxTime, bResetAlarm := "FVs_o/p".FV_4.bResetAlarm, bHaveFeedback := "FVs_o/p".FV_4.bCheckFeedback, bValveOpen => "FVs_o/p".FV_4.bOutOpen, iValveState => "FVs_o/p".FV_4.iOutState, bValveFault => "FVs_o/p".FV_4.bOutFault)
   END_RUNG
   // the same network as SCL:
   "FV_4"(bAuto_OpenCmd := "FVs_o/p".FV_4.bOpenCmd,   // "Valve(c/o)"
          bManualMode := "FVs_o/p".FV_4.bManualMode,
          bManualOpen := "FVs_o/p".FV_4.bManualOpen,
          bFeedbackOpen := "FVs_o/p".FV_4.bFeedbackOpen,
          tMaxTime := "FVs_o/p".FV_4.tMaxTime,
          bResetAlarm := "FVs_o/p".FV_4.bResetAlarm,
          bHaveFeedback := "FVs_o/p".FV_4.bCheckFeedback,
          bValveOpen => "FVs_o/p".FV_4.bOutOpen,
          iValveState => "FVs_o/p".FV_4.iOutState,
          bValveFault => "FVs_o/p".FV_4.bOutFault);
END_REGION

REGION Network 5: FV-5
   RUNG wire#powerrail
      "FV_5"(bAuto_OpenCmd := "FVs_o/p".FV_5.bOpenCmd, bManualMode := "FVs_o/p".FV_5.bManualMode, bManualOpen := "FVs_o/p".FV_5.bManualOpen, bFeedbackOpen := "FVs_o/p".FV_5.bFeedbackOpen, tMaxTime := "FVs_o/p".FV_5.tMaxTime, bResetAlarm := "FVs_o/p".FV_5.bResetAlarm, bHaveFeedback := "FVs_o/p".FV_5.bCheckFeedback, bValveOpen => "FVs_o/p".FV_5.bOutOpen, iValveState => "FVs_o/p".FV_5.iOutState, bValveFault => "FVs_o/p".FV_5.bOutFault)
   END_RUNG
   // the same network as SCL:
   "FV_5"(bAuto_OpenCmd := "FVs_o/p".FV_5.bOpenCmd,   // "Valve(c/o)"
          bManualMode := "FVs_o/p".FV_5.bManualMode,
          bManualOpen := "FVs_o/p".FV_5.bManualOpen,
          bFeedbackOpen := "FVs_o/p".FV_5.bFeedbackOpen,
          tMaxTime := "FVs_o/p".FV_5.tMaxTime,
          bResetAlarm := "FVs_o/p".FV_5.bResetAlarm,
          bHaveFeedback := "FVs_o/p".FV_5.bCheckFeedback,
          bValveOpen => "FVs_o/p".FV_5.bOutOpen,
          iValveState => "FVs_o/p".FV_5.iOutState,
          bValveFault => "FVs_o/p".FV_5.bOutFault);
END_REGION

REGION Network 6: FV-6
   RUNG wire#powerrail
      "FV_6"(bAuto_OpenCmd := "FVs_o/p".FV_6.bOpenCmd, bManualMode := "FVs_o/p".FV_6.bManualMode, bManualOpen := "FVs_o/p".FV_6.bManualOpen, bFeedbackOpen := "FVs_o/p".FV_6.bFeedbackOpen, tMaxTime := "FVs_o/p".FV_6.tMaxTime, bResetAlarm := "FVs_o/p".FV_6.bResetAlarm, bHaveFeedback := "FVs_o/p".FV_6.bCheckFeedback, bValveOpen => "FVs_o/p".FV_6.bOutOpen, iValveState => "FVs_o/p".FV_6.iOutState, bValveFault => "FVs_o/p".FV_6.bOutFault)
   END_RUNG
   // the same network as SCL:
   "FV_6"(bAuto_OpenCmd := "FVs_o/p".FV_6.bOpenCmd,   // "Valve(c/o)"
          bManualMode := "FVs_o/p".FV_6.bManualMode,
          bManualOpen := "FVs_o/p".FV_6.bManualOpen,
          bFeedbackOpen := "FVs_o/p".FV_6.bFeedbackOpen,
          tMaxTime := "FVs_o/p".FV_6.tMaxTime,
          bResetAlarm := "FVs_o/p".FV_6.bResetAlarm,
          bHaveFeedback := "FVs_o/p".FV_6.bCheckFeedback,
          bValveOpen => "FVs_o/p".FV_6.bOutOpen,
          iValveState => "FVs_o/p".FV_6.iOutState,
          bValveFault => "FVs_o/p".FV_6.bOutFault);
END_REGION

REGION Network 7: FV-7
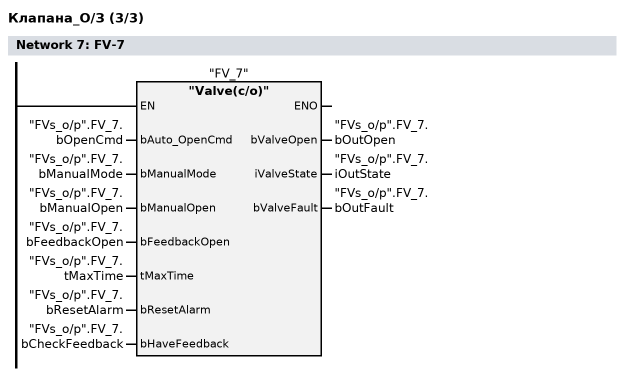
   RUNG wire#powerrail
      "FV_7"(bAuto_OpenCmd := "FVs_o/p".FV_7.bOpenCmd, bManualMode := "FVs_o/p".FV_7.bManualMode, bManualOpen := "FVs_o/p".FV_7.bManualOpen, bFeedbackOpen := "FVs_o/p".FV_7.bFeedbackOpen, tMaxTime := "FVs_o/p".FV_7.tMaxTime, bResetAlarm := "FVs_o/p".FV_7.bResetAlarm, bHaveFeedback := "FVs_o/p".FV_7.bCheckFeedback, bValveOpen => "FVs_o/p".FV_7.bOutOpen, iValveState => "FVs_o/p".FV_7.iOutState, bValveFault => "FVs_o/p".FV_7.bOutFault)
   END_RUNG
   // the same network as SCL:
   "FV_7"(bAuto_OpenCmd := "FVs_o/p".FV_7.bOpenCmd,   // "Valve(c/o)"
          bManualMode := "FVs_o/p".FV_7.bManualMode,
          bManualOpen := "FVs_o/p".FV_7.bManualOpen,
          bFeedbackOpen := "FVs_o/p".FV_7.bFeedbackOpen,
          tMaxTime := "FVs_o/p".FV_7.tMaxTime,
          bResetAlarm := "FVs_o/p".FV_7.bResetAlarm,
          bHaveFeedback := "FVs_o/p".FV_7.bCheckFeedback,
          bValveOpen => "FVs_o/p".FV_7.bOutOpen,
          iValveState => "FVs_o/p".FV_7.iOutState,
          bValveFault => "FVs_o/p".FV_7.bOutFault);
END_REGION
END_FUNCTION

FUNCTION "Клапана_Регул" : Void   // FC2, LAD
{ S7_Optimized_Access := 'TRUE' }
VERSION : 0.1
BEGIN

REGION Network 1: Клапан регулирующий - 1
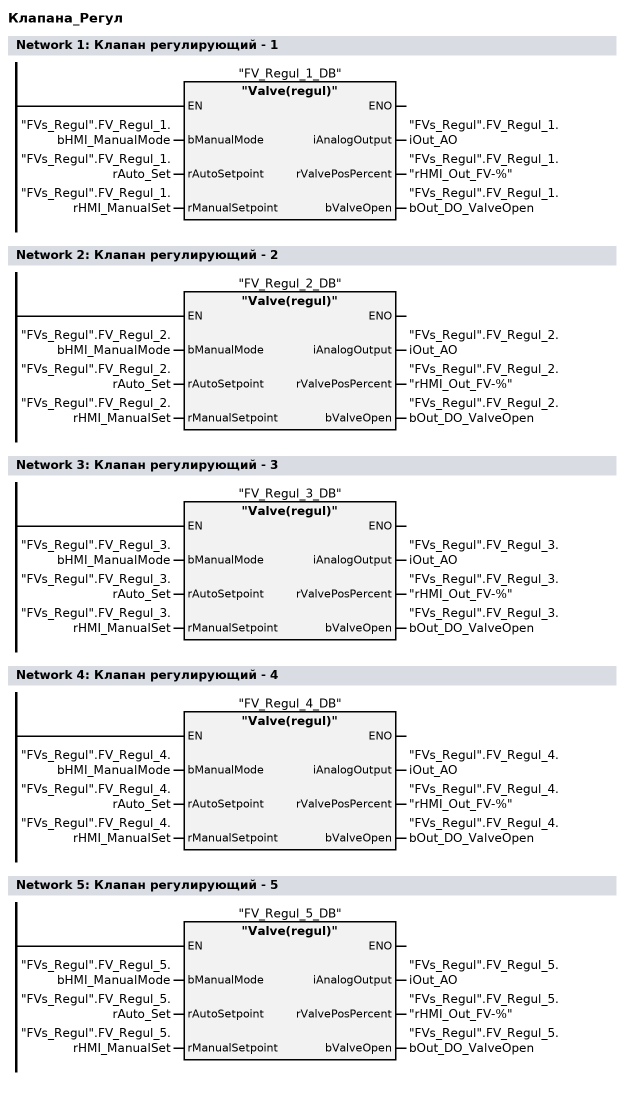
   RUNG wire#powerrail
      "FV_Regul_1_DB"(bManualMode := "FVs_Regul".FV_Regul_1.bHMI_ManualMode, rAutoSetpoint := "FVs_Regul".FV_Regul_1.rAuto_Set, rManualSetpoint := "FVs_Regul".FV_Regul_1.rHMI_ManualSet, iAnalogOutput => "FVs_Regul".FV_Regul_1.iOut_AO, rValvePosPercent => "FVs_Regul".FV_Regul_1."rHMI_Out_FV-%", bValveOpen => "FVs_Regul".FV_Regul_1.bOut_DO_ValveOpen)
   END_RUNG
   // the same network as SCL:
   "FV_Regul_1_DB"(bManualMode := "FVs_Regul".FV_Regul_1.bHMI_ManualMode,   // "Valve(regul)"
                   rAutoSetpoint := "FVs_Regul".FV_Regul_1.rAuto_Set,
                   rManualSetpoint := "FVs_Regul".FV_Regul_1.rHMI_ManualSet,
                   iAnalogOutput => "FVs_Regul".FV_Regul_1.iOut_AO,
                   rValvePosPercent => "FVs_Regul".FV_Regul_1."rHMI_Out_FV-%",
                   bValveOpen => "FVs_Regul".FV_Regul_1.bOut_DO_ValveOpen);
END_REGION

REGION Network 2: Клапан регулирующий - 2
   RUNG wire#powerrail
      "FV_Regul_2_DB"(bManualMode := "FVs_Regul".FV_Regul_2.bHMI_ManualMode, rAutoSetpoint := "FVs_Regul".FV_Regul_2.rAuto_Set, rManualSetpoint := "FVs_Regul".FV_Regul_2.rHMI_ManualSet, iAnalogOutput => "FVs_Regul".FV_Regul_2.iOut_AO, rValvePosPercent => "FVs_Regul".FV_Regul_2."rHMI_Out_FV-%", bValveOpen => "FVs_Regul".FV_Regul_2.bOut_DO_ValveOpen)
   END_RUNG
   // the same network as SCL:
   "FV_Regul_2_DB"(bManualMode := "FVs_Regul".FV_Regul_2.bHMI_ManualMode,   // "Valve(regul)"
                   rAutoSetpoint := "FVs_Regul".FV_Regul_2.rAuto_Set,
                   rManualSetpoint := "FVs_Regul".FV_Regul_2.rHMI_ManualSet,
                   iAnalogOutput => "FVs_Regul".FV_Regul_2.iOut_AO,
                   rValvePosPercent => "FVs_Regul".FV_Regul_2."rHMI_Out_FV-%",
                   bValveOpen => "FVs_Regul".FV_Regul_2.bOut_DO_ValveOpen);
END_REGION

REGION Network 3: Клапан регулирующий - 3
   RUNG wire#powerrail
      "FV_Regul_3_DB"(bManualMode := "FVs_Regul".FV_Regul_3.bHMI_ManualMode, rAutoSetpoint := "FVs_Regul".FV_Regul_3.rAuto_Set, rManualSetpoint := "FVs_Regul".FV_Regul_3.rHMI_ManualSet, iAnalogOutput => "FVs_Regul".FV_Regul_3.iOut_AO, rValvePosPercent => "FVs_Regul".FV_Regul_3."rHMI_Out_FV-%", bValveOpen => "FVs_Regul".FV_Regul_3.bOut_DO_ValveOpen)
   END_RUNG
   // the same network as SCL:
   "FV_Regul_3_DB"(bManualMode := "FVs_Regul".FV_Regul_3.bHMI_ManualMode,   // "Valve(regul)"
                   rAutoSetpoint := "FVs_Regul".FV_Regul_3.rAuto_Set,
                   rManualSetpoint := "FVs_Regul".FV_Regul_3.rHMI_ManualSet,
                   iAnalogOutput => "FVs_Regul".FV_Regul_3.iOut_AO,
                   rValvePosPercent => "FVs_Regul".FV_Regul_3."rHMI_Out_FV-%",
                   bValveOpen => "FVs_Regul".FV_Regul_3.bOut_DO_ValveOpen);
END_REGION

REGION Network 4: Клапан регулирующий - 4
   RUNG wire#powerrail
      "FV_Regul_4_DB"(bManualMode := "FVs_Regul".FV_Regul_4.bHMI_ManualMode, rAutoSetpoint := "FVs_Regul".FV_Regul_4.rAuto_Set, rManualSetpoint := "FVs_Regul".FV_Regul_4.rHMI_ManualSet, iAnalogOutput => "FVs_Regul".FV_Regul_4.iOut_AO, rValvePosPercent => "FVs_Regul".FV_Regul_4."rHMI_Out_FV-%", bValveOpen => "FVs_Regul".FV_Regul_4.bOut_DO_ValveOpen)
   END_RUNG
   // the same network as SCL:
   "FV_Regul_4_DB"(bManualMode := "FVs_Regul".FV_Regul_4.bHMI_ManualMode,   // "Valve(regul)"
                   rAutoSetpoint := "FVs_Regul".FV_Regul_4.rAuto_Set,
                   rManualSetpoint := "FVs_Regul".FV_Regul_4.rHMI_ManualSet,
                   iAnalogOutput => "FVs_Regul".FV_Regul_4.iOut_AO,
                   rValvePosPercent => "FVs_Regul".FV_Regul_4."rHMI_Out_FV-%",
                   bValveOpen => "FVs_Regul".FV_Regul_4.bOut_DO_ValveOpen);
END_REGION

REGION Network 5: Клапан регулирующий - 5
   RUNG wire#powerrail
      "FV_Regul_5_DB"(bManualMode := "FVs_Regul".FV_Regul_5.bHMI_ManualMode, rAutoSetpoint := "FVs_Regul".FV_Regul_5.rAuto_Set, rManualSetpoint := "FVs_Regul".FV_Regul_5.rHMI_ManualSet, iAnalogOutput => "FVs_Regul".FV_Regul_5.iOut_AO, rValvePosPercent => "FVs_Regul".FV_Regul_5."rHMI_Out_FV-%", bValveOpen => "FVs_Regul".FV_Regul_5.bOut_DO_ValveOpen)
   END_RUNG
   // the same network as SCL:
   "FV_Regul_5_DB"(bManualMode := "FVs_Regul".FV_Regul_5.bHMI_ManualMode,   // "Valve(regul)"
                   rAutoSetpoint := "FVs_Regul".FV_Regul_5.rAuto_Set,
                   rManualSetpoint := "FVs_Regul".FV_Regul_5.rHMI_ManualSet,
                   iAnalogOutput => "FVs_Regul".FV_Regul_5.iOut_AO,
                   rValvePosPercent => "FVs_Regul".FV_Regul_5."rHMI_Out_FV-%",
                   bValveOpen => "FVs_Regul".FV_Regul_5.bOut_DO_ValveOpen);
END_REGION
END_FUNCTION

FUNCTION "Зоны пастеризации_Контроль" : Void   // FC3, LAD
{ S7_Optimized_Access := 'TRUE' }
VERSION : 0.1
BEGIN

REGION Network 1: Зона 1
   // Зона 1 Преднагрев
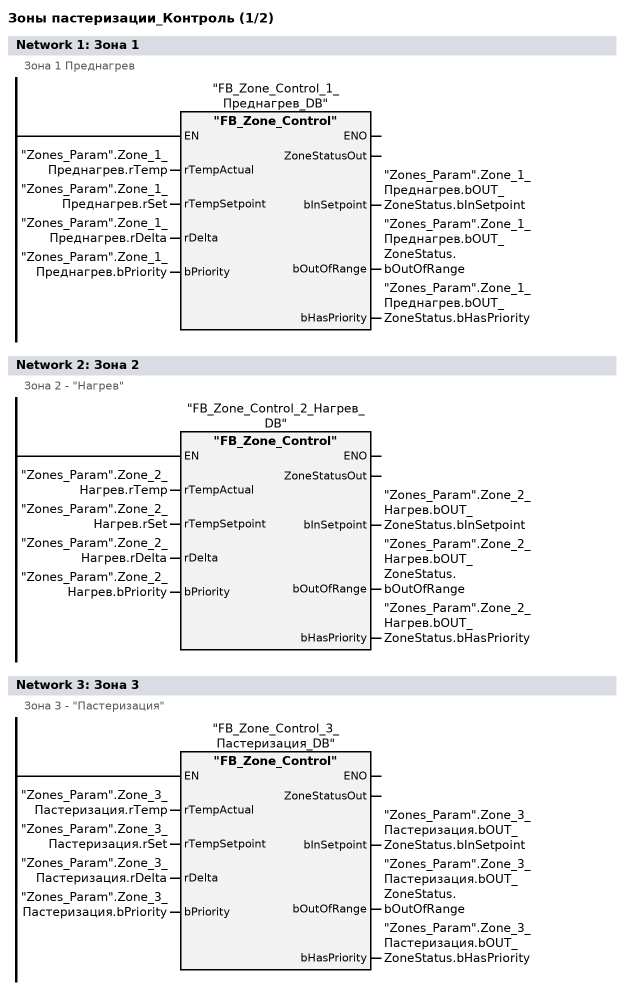
   RUNG wire#powerrail
      "FB_Zone_Control_1_Преднагрев_DB"(rTempActual := "Zones_Param".Zone_1_Преднагрев.rTemp, rTempSetpoint := "Zones_Param".Zone_1_Преднагрев.rSet, rDelta := "Zones_Param".Zone_1_Преднагрев.rDelta, bPriority := "Zones_Param".Zone_1_Преднагрев.bPriority, ZoneStatusOut =>, bInSetpoint => "Zones_Param".Zone_1_Преднагрев.bOUT_ZoneStatus.bInSetpoint, bOutOfRange => "Zones_Param".Zone_1_Преднагрев.bOUT_ZoneStatus.bOutOfRange, bHasPriority => "Zones_Param".Zone_1_Преднагрев.bOUT_ZoneStatus.bHasPriority)
   END_RUNG
   // the same network as SCL:
   "FB_Zone_Control_1_Преднагрев_DB"(rTempActual := "Zones_Param".Zone_1_Преднагрев.rTemp,   // "FB_Zone_Control"
                           rTempSetpoint := "Zones_Param".Zone_1_Преднагрев.rSet,
                           rDelta := "Zones_Param".Zone_1_Преднагрев.rDelta,
                           bPriority := "Zones_Param".Zone_1_Преднагрев.bPriority,
                           bInSetpoint => "Zones_Param".Zone_1_Преднагрев.bOUT_ZoneStatus.bInSetpoint,
                           bOutOfRange => "Zones_Param".Zone_1_Преднагрев.bOUT_ZoneStatus.bOutOfRange,
                           bHasPriority => "Zones_Param".Zone_1_Преднагрев.bOUT_ZoneStatus.bHasPriority);
END_REGION

REGION Network 2: Зона 2
   // Зона 2 - "Нагрев"
   RUNG wire#powerrail
      "FB_Zone_Control_2_Нагрев_DB"(rTempActual := "Zones_Param".Zone_2_Нагрев.rTemp, rTempSetpoint := "Zones_Param".Zone_2_Нагрев.rSet, rDelta := "Zones_Param".Zone_2_Нагрев.rDelta, bPriority := "Zones_Param".Zone_2_Нагрев.bPriority, ZoneStatusOut =>, bInSetpoint => "Zones_Param".Zone_2_Нагрев.bOUT_ZoneStatus.bInSetpoint, bOutOfRange => "Zones_Param".Zone_2_Нагрев.bOUT_ZoneStatus.bOutOfRange, bHasPriority => "Zones_Param".Zone_2_Нагрев.bOUT_ZoneStatus.bHasPriority)
   END_RUNG
   // the same network as SCL:
   "FB_Zone_Control_2_Нагрев_DB"(rTempActual := "Zones_Param".Zone_2_Нагрев.rTemp,   // "FB_Zone_Control"
                           rTempSetpoint := "Zones_Param".Zone_2_Нагрев.rSet,
                           rDelta := "Zones_Param".Zone_2_Нагрев.rDelta,
                           bPriority := "Zones_Param".Zone_2_Нагрев.bPriority,
                           bInSetpoint => "Zones_Param".Zone_2_Нагрев.bOUT_ZoneStatus.bInSetpoint,
                           bOutOfRange => "Zones_Param".Zone_2_Нагрев.bOUT_ZoneStatus.bOutOfRange,
                           bHasPriority => "Zones_Param".Zone_2_Нагрев.bOUT_ZoneStatus.bHasPriority);
END_REGION

REGION Network 3: Зона 3
   // Зона 3 - "Пастеризация"
   RUNG wire#powerrail
      "FB_Zone_Control_3_Пастеризация_DB"(rTempActual := "Zones_Param".Zone_3_Пастеризация.rTemp, rTempSetpoint := "Zones_Param".Zone_3_Пастеризация.rSet, rDelta := "Zones_Param".Zone_3_Пастеризация.rDelta, bPriority := "Zones_Param".Zone_3_Пастеризация.bPriority, ZoneStatusOut =>, bInSetpoint => "Zones_Param".Zone_3_Пастеризация.bOUT_ZoneStatus.bInSetpoint, bOutOfRange => "Zones_Param".Zone_3_Пастеризация.bOUT_ZoneStatus.bOutOfRange, bHasPriority => "Zones_Param".Zone_3_Пастеризация.bOUT_ZoneStatus.bHasPriority)
   END_RUNG
   // the same network as SCL:
   "FB_Zone_Control_3_Пастеризация_DB"(rTempActual := "Zones_Param".Zone_3_Пастеризация.rTemp,   // "FB_Zone_Control"
                           rTempSetpoint := "Zones_Param".Zone_3_Пастеризация.rSet,
                           rDelta := "Zones_Param".Zone_3_Пастеризация.rDelta,
                           bPriority := "Zones_Param".Zone_3_Пастеризация.bPriority,
                           bInSetpoint => "Zones_Param".Zone_3_Пастеризация.bOUT_ZoneStatus.bInSetpoint,
                           bOutOfRange => "Zones_Param".Zone_3_Пастеризация.bOUT_ZoneStatus.bOutOfRange,
                           bHasPriority => "Zones_Param".Zone_3_Пастеризация.bOUT_ZoneStatus.bHasPriority);
END_REGION

REGION Network 4: Зона 4
   // Зона 4 - "Охлаждение 1"
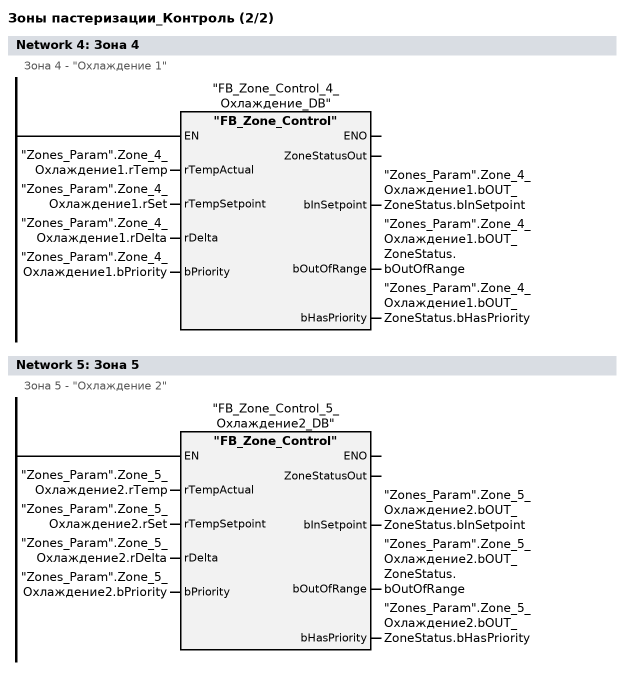
   RUNG wire#powerrail
      "FB_Zone_Control_4_Охлаждение_DB"(rTempActual := "Zones_Param".Zone_4_Охлаждение1.rTemp, rTempSetpoint := "Zones_Param".Zone_4_Охлаждение1.rSet, rDelta := "Zones_Param".Zone_4_Охлаждение1.rDelta, bPriority := "Zones_Param".Zone_4_Охлаждение1.bPriority, ZoneStatusOut =>, bInSetpoint => "Zones_Param".Zone_4_Охлаждение1.bOUT_ZoneStatus.bInSetpoint, bOutOfRange => "Zones_Param".Zone_4_Охлаждение1.bOUT_ZoneStatus.bOutOfRange, bHasPriority => "Zones_Param".Zone_4_Охлаждение1.bOUT_ZoneStatus.bHasPriority)
   END_RUNG
   // the same network as SCL:
   "FB_Zone_Control_4_Охлаждение_DB"(rTempActual := "Zones_Param".Zone_4_Охлаждение1.rTemp,   // "FB_Zone_Control"
                           rTempSetpoint := "Zones_Param".Zone_4_Охлаждение1.rSet,
                           rDelta := "Zones_Param".Zone_4_Охлаждение1.rDelta,
                           bPriority := "Zones_Param".Zone_4_Охлаждение1.bPriority,
                           bInSetpoint => "Zones_Param".Zone_4_Охлаждение1.bOUT_ZoneStatus.bInSetpoint,
                           bOutOfRange => "Zones_Param".Zone_4_Охлаждение1.bOUT_ZoneStatus.bOutOfRange,
                           bHasPriority => "Zones_Param".Zone_4_Охлаждение1.bOUT_ZoneStatus.bHasPriority);
END_REGION

REGION Network 5: Зона 5
   // Зона 5 - "Охлаждение 2"
   RUNG wire#powerrail
      "FB_Zone_Control_5_Охлаждение2_DB"(rTempActual := "Zones_Param".Zone_5_Охлаждение2.rTemp, rTempSetpoint := "Zones_Param".Zone_5_Охлаждение2.rSet, rDelta := "Zones_Param".Zone_5_Охлаждение2.rDelta, bPriority := "Zones_Param".Zone_5_Охлаждение2.bPriority, ZoneStatusOut =>, bInSetpoint => "Zones_Param".Zone_5_Охлаждение2.bOUT_ZoneStatus.bInSetpoint, bOutOfRange => "Zones_Param".Zone_5_Охлаждение2.bOUT_ZoneStatus.bOutOfRange, bHasPriority => "Zones_Param".Zone_5_Охлаждение2.bOUT_ZoneStatus.bHasPriority)
   END_RUNG
   // the same network as SCL:
   "FB_Zone_Control_5_Охлаждение2_DB"(rTempActual := "Zones_Param".Zone_5_Охлаждение2.rTemp,   // "FB_Zone_Control"
                           rTempSetpoint := "Zones_Param".Zone_5_Охлаждение2.rSet,
                           rDelta := "Zones_Param".Zone_5_Охлаждение2.rDelta,
                           bPriority := "Zones_Param".Zone_5_Охлаждение2.bPriority,
                           bInSetpoint => "Zones_Param".Zone_5_Охлаждение2.bOUT_ZoneStatus.bInSetpoint,
                           bOutOfRange => "Zones_Param".Zone_5_Охлаждение2.bOUT_ZoneStatus.bOutOfRange,
                           bHasPriority => "Zones_Param".Zone_5_Охлаждение2.bOUT_ZoneStatus.bHasPriority);
END_REGION
END_FUNCTION

FUNCTION "Аварии" : Void   // FC4, LAD
{ S7_Optimized_Access := 'TRUE' }
VERSION : 0.1
   VAR_OUTPUT
      xAlarm : Bool;   // Есть активные аварии
   END_VAR
BEGIN

REGION Network 1
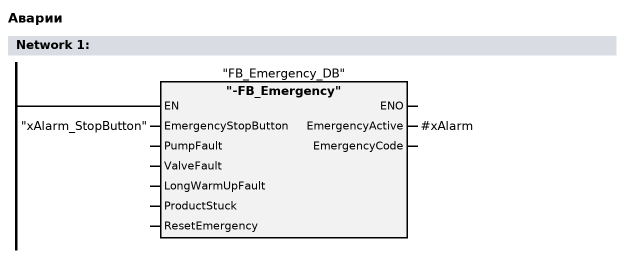
   RUNG wire#powerrail
      "FB_Emergency_DB"(EmergencyStopButton := "xAlarm_StopButton", PumpFault :=, ValveFault :=, LongWarmUpFault :=, ProductStuck :=, ResetEmergency :=, EmergencyActive => #xAlarm, EmergencyCode =>)
   END_RUNG
   // the same network as SCL:
   "FB_Emergency_DB"(EmergencyStopButton := "xAlarm_StopButton", EmergencyActive => #xAlarm);   // "-FB_Emergency"
END_REGION

REGION Network 3 (SCL): Есть активные аварии
END_REGION
END_FUNCTION

ORGANIZATION_BLOCK "Main"   // OB1, LAD, ProgramCycle
TITLE = "Основкая программа"
{ S7_Optimized_Access := 'TRUE' }
VERSION : 0.1
BEGIN

REGION Network 1: Аварии
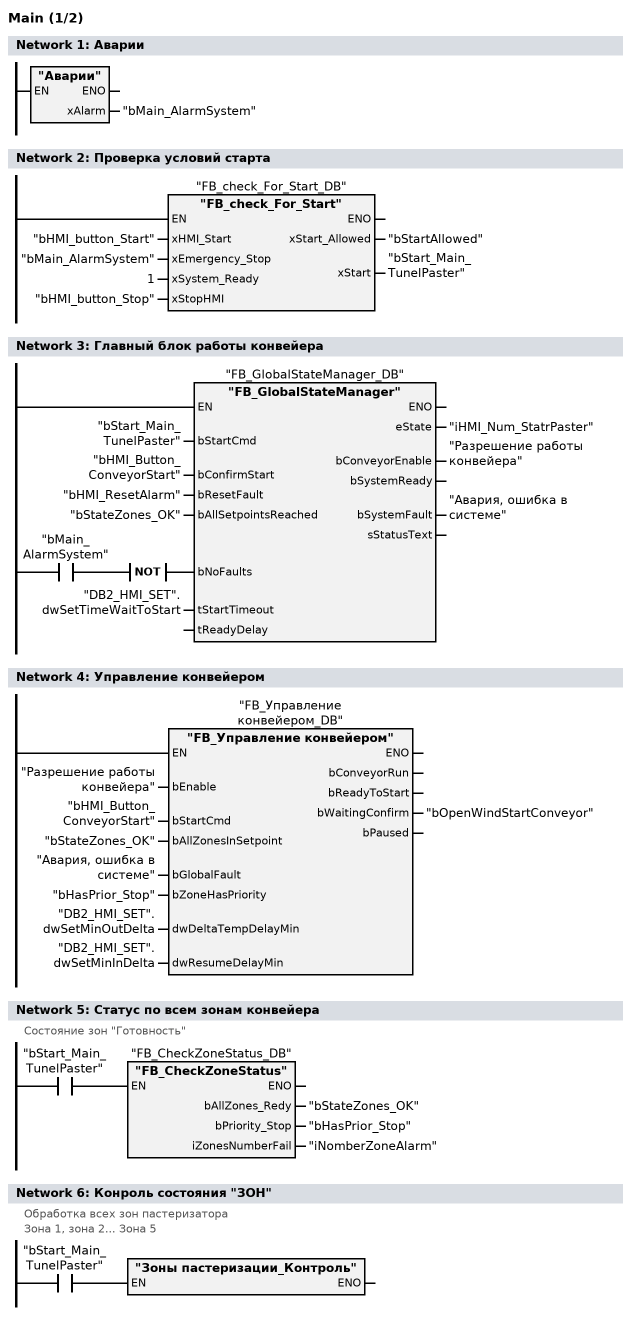
   RUNG wire#powerrail
      "Аварии"(xAlarm => "bMain_AlarmSystem")
   END_RUNG
   // the same network as SCL:
   "Аварии"(xAlarm => "bMain_AlarmSystem");
END_REGION

REGION Network 2: Проверка условий старта
   RUNG wire#powerrail
      "FB_check_For_Start_DB"(xHMI_Start := "bHMI_button_Start", xEmergency_Stop := "bMain_AlarmSystem", xSystem_Ready := 1, xStopHMI := "bHMI_button_Stop", xStart_Allowed => "bStartAllowed", xStart => "bStart_Main_TunelPaster")
   END_RUNG
   // the same network as SCL:
   "FB_check_For_Start_DB"(xHMI_Start := "bHMI_button_Start",   // "FB_check_For_Start"
                           xEmergency_Stop := "bMain_AlarmSystem",
                           xSystem_Ready := 1,
                           xStopHMI := "bHMI_button_Stop",
                           xStart_Allowed => "bStartAllowed",
                           xStart => "bStart_Main_TunelPaster");
END_REGION

REGION Network 3: Главный блок работы конвейера
   RUNG wire#powerrail
      "FB_GlobalStateManager_DB"(bNoFaults := wire#w1, bStartCmd := "bStart_Main_TunelPaster", bConfirmStart := "bHMI_Button_ConveyorStart", bResetFault := "bHMI_ResetAlarm", bAllSetpointsReached := "bStateZones_OK", tStartTimeout := "DB2_HMI_SET".dwSetTimeWaitToStart, tReadyDelay :=, eState => "iHMI_Num_StatrPaster", bConveyorEnable => "Разрешение работы конвейера", bSystemReady =>, bSystemFault => "Авария, ошибка в системе", sStatusText =>)
   END_RUNG
   RUNG wire#powerrail
      Contact( "bMain_AlarmSystem" )
      Not()
   END_RUNG wire#w1
   // the same network as SCL:
   "FB_GlobalStateManager_DB"(bStartCmd := "bStart_Main_TunelPaster",   // "FB_GlobalStateManager"
                           bConfirmStart := "bHMI_Button_ConveyorStart",
                           bResetFault := "bHMI_ResetAlarm",
                           bAllSetpointsReached := "bStateZones_OK",
                           bNoFaults := NOT "bMain_AlarmSystem",
                           tStartTimeout := "DB2_HMI_SET".dwSetTimeWaitToStart,
                           eState => "iHMI_Num_StatrPaster",
                           bConveyorEnable => "Разрешение работы конвейера",
                           bSystemFault => "Авария, ошибка в системе");
END_REGION

REGION Network 4: Управление конвейером
   RUNG wire#powerrail
      "FB_Управление конвейером_DB"(bEnable := "Разрешение работы конвейера", bStartCmd := "bHMI_Button_ConveyorStart", bAllZonesInSetpoint := "bStateZones_OK", bGlobalFault := "Авария, ошибка в системе", bZoneHasPriority := "bHasPrior_Stop", dwDeltaTempDelayMin := "DB2_HMI_SET".dwSetMinOutDelta, dwResumeDelayMin := "DB2_HMI_SET".dwSetMinInDelta, bConveyorRun =>, bReadyToStart =>, bWaitingConfirm => "bOpenWindStartConveyor", bPaused =>)
   END_RUNG
   // the same network as SCL:
   "FB_Управление конвейером_DB"(bEnable := "Разрешение работы конвейера",   // "FB_Управление конвейером"
                           bStartCmd := "bHMI_Button_ConveyorStart",
                           bAllZonesInSetpoint := "bStateZones_OK",
                           bGlobalFault := "Авария, ошибка в системе",
                           bZoneHasPriority := "bHasPrior_Stop",
                           dwDeltaTempDelayMin := "DB2_HMI_SET".dwSetMinOutDelta,
                           dwResumeDelayMin := "DB2_HMI_SET".dwSetMinInDelta,
                           bWaitingConfirm => "bOpenWindStartConveyor");
END_REGION

REGION Network 5: Статус по всем зонам конвейера
   // Состояние зон "Готовность"
   RUNG wire#powerrail
      Contact( "bStart_Main_TunelPaster" )
      "FB_CheckZoneStatus_DB"(bAllZones_Redy => "bStateZones_OK", bPriority_Stop => "bHasPrior_Stop", iZonesNumberFail => "iNomberZoneAlarm")
   END_RUNG
   // the same network as SCL:
   IF "bStart_Main_TunelPaster" THEN
       "FB_CheckZoneStatus_DB"(bAllZones_Redy => "bStateZones_OK",   // "FB_CheckZoneStatus"
                               bPriority_Stop => "bHasPrior_Stop",
                               iZonesNumberFail => "iNomberZoneAlarm");
   END_IF;
END_REGION

REGION Network 6: Конроль состояния "ЗОН"
   // Обработка всех зон пастеризатора
   // Зона 1, зона 2... Зона 5
   RUNG wire#powerrail
      Contact( "bStart_Main_TunelPaster" )
      "Зоны пастеризации_Контроль"()
   END_RUNG
   // the same network as SCL:
   IF "bStart_Main_TunelPaster" THEN "Зоны пастеризации_Контроль"(); END_IF;
END_REGION

REGION Network 7: Расчет PE и скорости конвейера
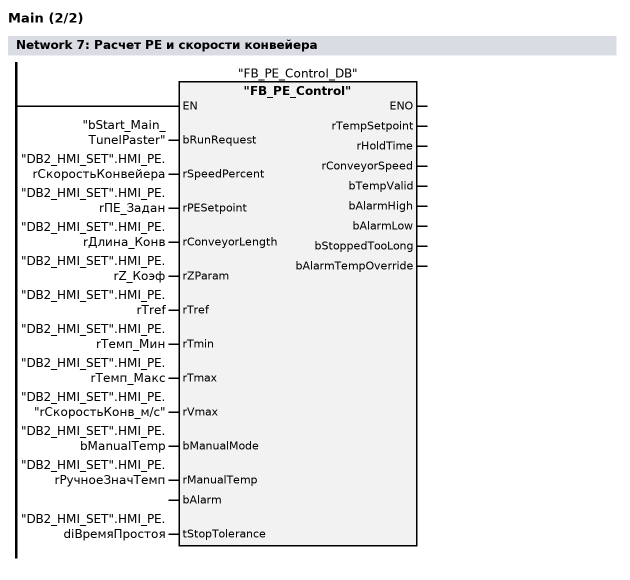
   RUNG wire#powerrail
      "FB_PE_Control_DB"(bRunRequest := "bStart_Main_TunelPaster", rSpeedPercent := "DB2_HMI_SET".HMI_PE.rСкоростьКонвейера, rPESetpoint := "DB2_HMI_SET".HMI_PE.rПЕ_Задан, rConveyorLength := "DB2_HMI_SET".HMI_PE.rДлина_Конв, rZParam := "DB2_HMI_SET".HMI_PE.rZ_Коэф, rTref := "DB2_HMI_SET".HMI_PE.rТref, rTmin := "DB2_HMI_SET".HMI_PE.rТемп_Мин, rTmax := "DB2_HMI_SET".HMI_PE.rТемп_Макс, rVmax := "DB2_HMI_SET".HMI_PE."rСкоростьКонв_м/с", bManualMode := "DB2_HMI_SET".HMI_PE.bManualTemp, rManualTemp := "DB2_HMI_SET".HMI_PE.rРучноеЗначТемп, bAlarm :=, tStopTolerance := "DB2_HMI_SET".HMI_PE.diВремяПростоя, rTempSetpoint =>, rHoldTime =>, rConveyorSpeed =>, bTempValid =>, bAlarmHigh =>, bAlarmLow =>, bStoppedTooLong =>, bAlarmTempOverride =>)
   END_RUNG
   // the same network as SCL:
   "FB_PE_Control_DB"(bRunRequest := "bStart_Main_TunelPaster",   // "FB_PE_Control"
                      rSpeedPercent := "DB2_HMI_SET".HMI_PE.rСкоростьКонвейера,
                      rPESetpoint := "DB2_HMI_SET".HMI_PE.rПЕ_Задан,
                      rConveyorLength := "DB2_HMI_SET".HMI_PE.rДлина_Конв,
                      rZParam := "DB2_HMI_SET".HMI_PE.rZ_Коэф,
                      rTref := "DB2_HMI_SET".HMI_PE.rТref,
                      rTmin := "DB2_HMI_SET".HMI_PE.rТемп_Мин,
                      rTmax := "DB2_HMI_SET".HMI_PE.rТемп_Макс,
                      rVmax := "DB2_HMI_SET".HMI_PE."rСкоростьКонв_м/с",
                      bManualMode := "DB2_HMI_SET".HMI_PE.bManualTemp,
                      rManualTemp := "DB2_HMI_SET".HMI_PE.rРучноеЗначТемп,
                      tStopTolerance := "DB2_HMI_SET".HMI_PE.diВремяПростоя);
END_REGION
END_ORGANIZATION_BLOCK

ORGANIZATION_BLOCK "PID"   // OB30, LAD, CyclicInterrupt
{ S7_Optimized_Access := 'TRUE' }
VERSION : 0.1
   VAR_INPUT
      Initial_Call : Bool;   // Initial call of this OB
      Event_Count : Int;   // Events discarded
   END_VAR
BEGIN

REGION Network 1: ПИД - Зона 1
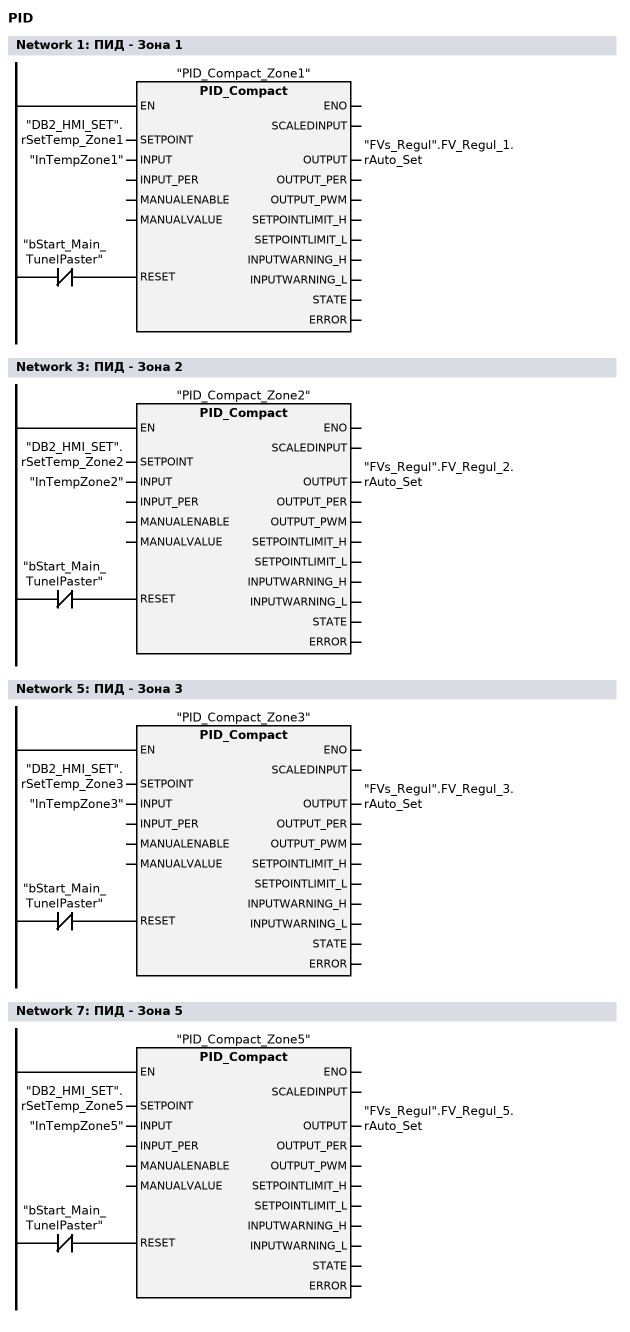
   "PID_Compact_Zone1"(Setpoint := "DB2_HMI_SET".rSetTemp_Zone1,   // PID_Compact
                       Input := "InTempZone1",
                       Reset := NOT "bStart_Main_TunelPaster",
                       Output => "FVs_Regul".FV_Regul_1.rAuto_Set);
END_REGION

REGION Network 2 (SCL): Выбор типа ПИД - Зона 1
   // 0 - Нагрев; 1 - Охлаждение
   "PID_Compact_Zone1".sPid_Cmpt.b_InvCtrl := "bTypePID_Zone1";
   (*
   "PID_Compact_Zone1".sRet.r_Ctrl_Gain := "DB2_HMI_SET".k_PID_Zona1.Gain; // Изменение коэф. П
   "PID_Compact_Zone1".sRet.r_Ctrl_Ti  := "DB2_HMI_SET".k_PID_Zona1.I; // Изменение коэф И
   "PID_Compact_Zone1".sRet.r_Ctrl_Td  := "DB2_HMI_SET".k_PID_Zona1.D; // Изменение коэф Д
   *)
END_REGION

REGION Network 3: ПИД - Зона 2
   "PID_Compact_Zone2"(Setpoint := "DB2_HMI_SET".rSetTemp_Zone2,   // PID_Compact
                       Input := "InTempZone2",
                       Reset := NOT "bStart_Main_TunelPaster",
                       Output => "FVs_Regul".FV_Regul_2.rAuto_Set);
END_REGION

REGION Network 4 (SCL): Выбор типа ПИД Зона 2
   // 0 - Нагрев; 1 - Охлаждение
   "PID_Compact_Zone2".sPid_Cmpt.b_InvCtrl := "bTypePID_Zone2";
END_REGION

REGION Network 5: ПИД - Зона 3
   "PID_Compact_Zone3"(Setpoint := "DB2_HMI_SET".rSetTemp_Zone3,   // PID_Compact
                       Input := "InTempZone3",
                       Reset := NOT "bStart_Main_TunelPaster",
                       Output => "FVs_Regul".FV_Regul_3.rAuto_Set);
END_REGION

REGION Network 6 (SCL): Выбор типа ПИД Зона 4
   // 0 - Нагрев; 1 - Охлаждение
   "PID_Compact_Zone3".sPid_Cmpt.b_InvCtrl := "bTypePID_Zone3";
END_REGION

REGION Network 7: ПИД - Зона 5
   "PID_Compact_Zone5"(Setpoint := "DB2_HMI_SET".rSetTemp_Zone5,   // PID_Compact
                       Input := "InTempZone5",
                       Reset := NOT "bStart_Main_TunelPaster",
                       Output => "FVs_Regul".FV_Regul_5.rAuto_Set);
END_REGION

REGION Network 8 (SCL): Выбор типа ПИД Зона 4
   // 0 - Нагрев; 1 - Охлаждение
   "PID_Compact_Zone5".sPid_Cmpt.b_InvCtrl := "bTypePID_Zone5";
END_REGION
END_ORGANIZATION_BLOCK

ORGANIZATION_BLOCK "Работа устройств"   // OB123, LAD, ProgramCycle
TITLE = Работа физических устройств
{ S7_Optimized_Access := 'TRUE' }
VERSION : 0.1
// Насосы, клапана, и т.д.
   VAR_INPUT
      Initial_Call : Bool;   // Initial call of this OB
      Remanence : Bool;   // =True, if remanent data are available
   END_VAR
BEGIN

REGION Network 1: Клапана Открыт/Закрыт
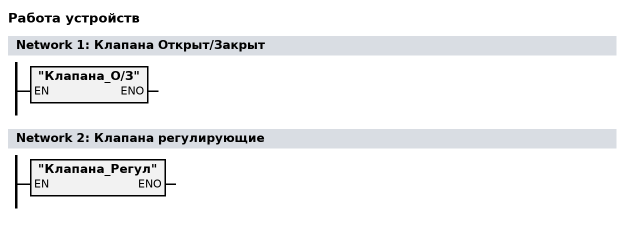
   RUNG wire#powerrail
      "Клапана_О/З"()
   END_RUNG
   // the same network as SCL:
   "Клапана_О/З"();
END_REGION

REGION Network 2: Клапана регулирующие
   RUNG wire#powerrail
      "Клапана_Регул"()
   END_RUNG
   // the same network as SCL:
   "Клапана_Регул"();
END_REGION

REGION Network 3: Насосы (старт/стоп)
END_REGION

REGION Network 4: Насосы (частотник)
END_REGION

REGION Network 5: Мотор конвейера
END_REGION
END_ORGANIZATION_BLOCK

ORGANIZATION_BLOCK "Test_SCL"   // OB124, SCL, ProgramCycle
TITLE = "Main Program Sweep (Cycle)"
{ S7_Optimized_Access := 'TRUE' }
VERSION : 0.1
   VAR_INPUT
      Initial_Call : Bool;   // Initial call of this OB
      Remanence : Bool;   // =True, if remanent data are available
   END_VAR
BEGIN
END_ORGANIZATION_BLOCK

// folder: Насосы

FUNCTION "Насосы" : Void   // FC5, LAD
{ S7_Optimized_Access := 'TRUE' }
VERSION : 0.1
BEGIN

REGION Network 1
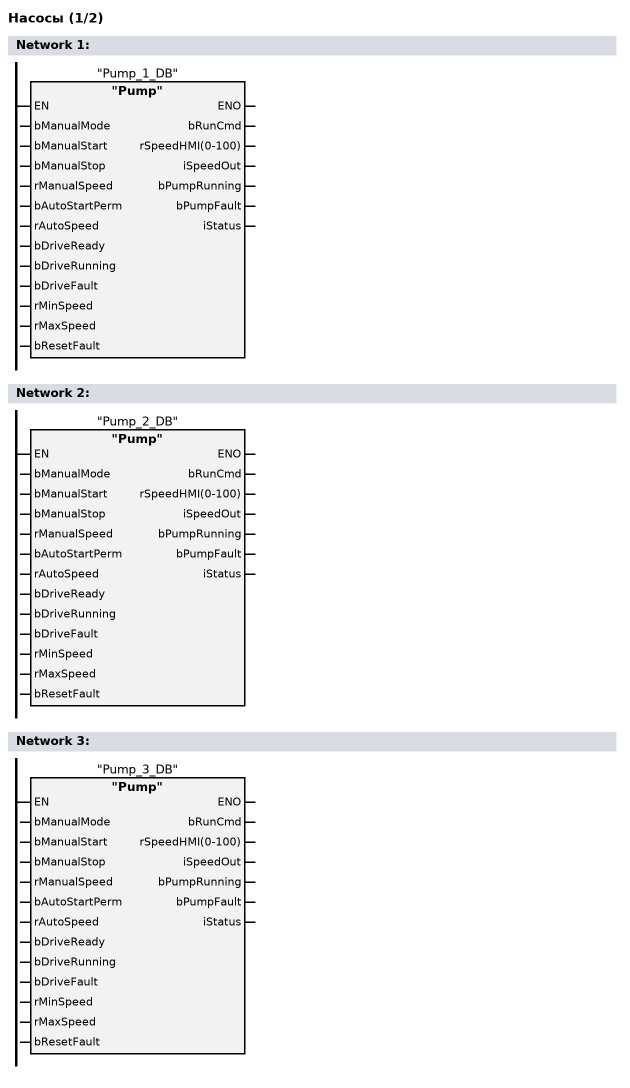
   RUNG wire#powerrail
      "Pump_1_DB"(bManualMode :=, bManualStart :=, bManualStop :=, rManualSpeed :=, bAutoStartPerm :=, rAutoSpeed :=, bDriveReady :=, bDriveRunning :=, bDriveFault :=, rMinSpeed :=, rMaxSpeed :=, bResetFault :=, bRunCmd =>, "rSpeedHMI(0-100)" =>, iSpeedOut =>, bPumpRunning =>, bPumpFault =>, iStatus =>)
   END_RUNG
   // the same network as SCL:
   "Pump_1_DB"();   // "Pump"
END_REGION

REGION Network 2
   RUNG wire#powerrail
      "Pump_2_DB"(bManualMode :=, bManualStart :=, bManualStop :=, rManualSpeed :=, bAutoStartPerm :=, rAutoSpeed :=, bDriveReady :=, bDriveRunning :=, bDriveFault :=, rMinSpeed :=, rMaxSpeed :=, bResetFault :=, bRunCmd =>, "rSpeedHMI(0-100)" =>, iSpeedOut =>, bPumpRunning =>, bPumpFault =>, iStatus =>)
   END_RUNG
   // the same network as SCL:
   "Pump_2_DB"();   // "Pump"
END_REGION

REGION Network 3
   RUNG wire#powerrail
      "Pump_3_DB"(bManualMode :=, bManualStart :=, bManualStop :=, rManualSpeed :=, bAutoStartPerm :=, rAutoSpeed :=, bDriveReady :=, bDriveRunning :=, bDriveFault :=, rMinSpeed :=, rMaxSpeed :=, bResetFault :=, bRunCmd =>, "rSpeedHMI(0-100)" =>, iSpeedOut =>, bPumpRunning =>, bPumpFault =>, iStatus =>)
   END_RUNG
   // the same network as SCL:
   "Pump_3_DB"();   // "Pump"
END_REGION

REGION Network 4
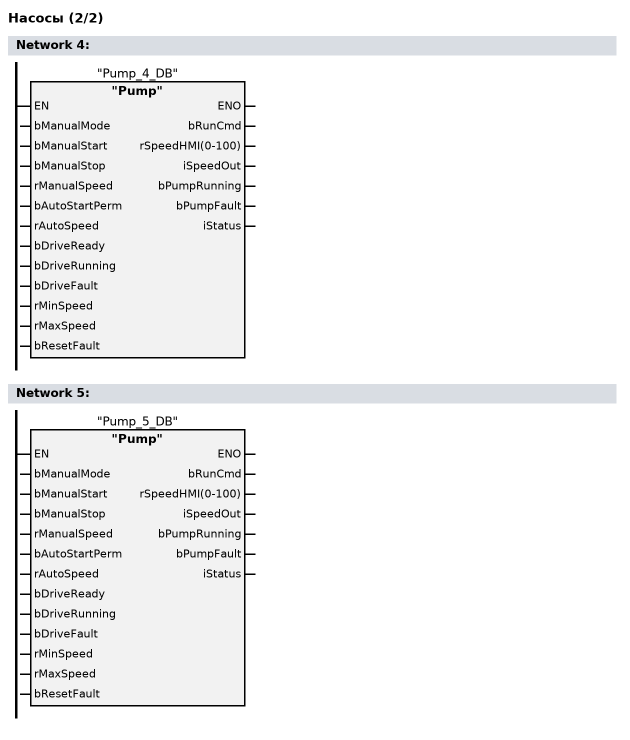
   RUNG wire#powerrail
      "Pump_4_DB"(bManualMode :=, bManualStart :=, bManualStop :=, rManualSpeed :=, bAutoStartPerm :=, rAutoSpeed :=, bDriveReady :=, bDriveRunning :=, bDriveFault :=, rMinSpeed :=, rMaxSpeed :=, bResetFault :=, bRunCmd =>, "rSpeedHMI(0-100)" =>, iSpeedOut =>, bPumpRunning =>, bPumpFault =>, iStatus =>)
   END_RUNG
   // the same network as SCL:
   "Pump_4_DB"();   // "Pump"
END_REGION

REGION Network 5
   RUNG wire#powerrail
      "Pump_5_DB"(bManualMode :=, bManualStart :=, bManualStop :=, rManualSpeed :=, bAutoStartPerm :=, rAutoSpeed :=, bDriveReady :=, bDriveRunning :=, bDriveFault :=, rMinSpeed :=, rMaxSpeed :=, bResetFault :=, bRunCmd =>, "rSpeedHMI(0-100)" =>, iSpeedOut =>, bPumpRunning =>, bPumpFault =>, iStatus =>)
   END_RUNG
   // the same network as SCL:
   "Pump_5_DB"();   // "Pump"
END_REGION
END_FUNCTION